// TwinCAT 3 PLC project Projet_Base
// ProgramVersion: 3.1.4022.3
// libraries:
//   Tc2_ControllerToolbox, * (Beckhoff Automation GmbH)
//   Tc2_IEC60870_5_10x, * (Beckhoff Automation GmbH)
//   Tc2_ModbusRTU, * (Beckhoff Automation GmbH)
//   Tc2_ModbusSrv, * (Beckhoff Automation GmbH)
//   Tc2_SerialCom, * (Beckhoff Automation GmbH)
//   Tc2_Standard, * (Beckhoff Automation GmbH)
//   Tc2_System, * (Beckhoff Automation GmbH)
//   Tc2_TcpIp, * (Beckhoff Automation GmbH)
//   Tc2_Utilities, * (Beckhoff Automation GmbH)
//   Tc3_Database, * (Beckhoff Automation GmbH)
//   Tc3_Module, * (Beckhoff Automation GmbH)
// project tree:
//   00_FunctionsBlocks/Beckhoff/AlarmManagement/ FB_HeartBeatMasterBackup.TcPOU (not stored), FUN_Alarms_CSV.TcPOU, FUN_ReadAlarm_CSV.TcPOU (not stored), ServerCSV.TcDUT, ServerSms.TcDUT, SMS_Server.TcPOU
//   00_FunctionsBlocks/Beckhoff/Annexesfunction/ FB_RestartService.TcPOU, FUN_ConnectVPN.TcPOU (not stored), FUN_DisconnectVPN.TcPOU (not stored), FUN_GetPublicIp.TcPOU (not stored), FUN_PingHost.TcPOU (not stored), PRG_RestartPlc.TcPOU (not stored)
//   00_FunctionsBlocks/Beckhoff/Communication/IEC104/ E_ComState.TcDUT (not stored), FB_IEC104ServerAkuo.TcPOU (not stored), GVL_Cst.TcGVL (not stored), ST_IEC104AkuoParam.TcDUT (not stored)
//   00_FunctionsBlocks/Beckhoff/Communication/Mail/ FUN_SendMail.TcPOU, ServerMail.TcDUT
//   00_FunctionsBlocks/Beckhoff/Communication/ModbusRTU/ CheckStruct.TcPOU (not stored), FB_ModbusRTU.TcPOU (not stored), FB_ReadModbusRTU_V2.TcPOU (not stored), Sample_ModbusRTU.TcPOU (not stored), Struct_InputRTU.TcDUT (not stored)
//   00_FunctionsBlocks/Beckhoff/Communication/ModbusTCP/ FB_ModbusRead.TcPOU (not stored), FB_ModbusReadCoils.TcPOU (not stored), FB_ModbusReadInput.TcPOU (not stored), FB_ModbusReadInputRegs.TcPOU (not stored), FB_ModbusWrite.TcPOU (not stored), FB_ModbusWriteMultipleCoils.TcPOU (not stored), FB_ModbusWriteSingleCoil.TcPOU (not stored), FB_ModbusWriteSingleRegister.TcPOU (not stored)
//   00_FunctionsBlocks/Beckhoff/Communication/SMS/ FB_DeleteAllSMS.TcPOU (not stored), FB_DeleteSMS.TcPOU (not stored), FB_Extract_Num_Mes.TcPOU (not stored), FB_Login.TcPOU (not stored), FB_ReadSMS.TcPOU (not stored), FB_SendSMS.TcPOU (not stored), ST_SMSDataSetEntry_Read.TcDUT (not stored), ST_SMSDataSetEntry_Send.TcDUT (not stored)
//   00_FunctionsBlocks/Beckhoff/Database/ CheckConfig.TcPOU (not stored), PRG_EpochConverter.TcPOU (not stored), PRG_TimestructConverter.TcPOU (not stored), St_DataHisto.TcDUT (not stored), St_DataHisto_Epoch.TcDUT (not stored), UnixTimestamp.TcPOU (not stored)
//   00_FunctionsBlocks/Beckhoff/Database/Firebird/ Firebird_CreateTables.TcPOU (not stored), Firebird_InsertBuffer.TcPOU (not stored), Firebird_InsertBuffer_vEpoch.TcPOU (not stored), Firebird_ReadAlarms.TcPOU (not stored), Firebird_RetrieveHDBID.TcPOU (not stored), Firebird_SelectBuffer.TcPOU (not stored), Firebird_WriteAlarms.TcPOU (not stored), LoggerFirebird.TcDUT (not stored), St_AlarmsV2.TcDUT (not stored)
//   00_FunctionsBlocks/Beckhoff/Database/InfluxDb/ InfluxDb_AlarmsManagement.TcPOU (not stored), InfluxDb_ReadValues.TcPOU (not stored), InfluxDb_WriteAlarms.TcPOU (not stored), InfluxDb_WriteStruct.TcPOU (not stored), LoggerInfluxDb.TcDUT (not stored), ST_InfluxAlarmsInsert.TcDUT (not stored), ST_InfluxAlarmsRetrieve.TcDUT (not stored)
//   00_FunctionsBlocks/Beckhoff/Database/SQLCe/ FB_SQLExpert_InsertBuffer_1.TcPOU (not stored)
//   00_FunctionsBlocks/Beckhoff/Database/SQLite/ SQLite_CreateDb_V2_1.TcPOU (not stored), SQLite_DeleteConfDb_1.TcPOU (not stored)
//   00_FunctionsBlocks/Beckhoff/DataProcessing/Compress/ FB_CompressFile.TcPOU (not stored), FUN_CompressCSV.TcPOU (not stored)
//   00_FunctionsBlocks/Beckhoff/DataProcessing/Database/ DataBase_V2.TcPOU (not stored), FB_DeleteFile.TcPOU (not stored), FB_SQLExpert_InsertBuffer.TcPOU (not stored), SQLite_CreateDb_V2.TcPOU (not stored), SQLite_DeleteConfDb.TcPOU (not stored)
//   00_FunctionsBlocks/Beckhoff/DataProcessing/ FB_MergeWordsToFloat.TcPOU (not stored), FB_MessageDynamique.TcPOU (not stored), FB_SplitFloatToWords.TcPOU (not stored), FB_WordsToFloat32MLE.TcPOU (not stored), FUN_Transpose.TcPOU (not stored), MOYENNE.TcPOU (not stored), ReplaceAll.TcPOU (not stored), SavePersistent.TcPOU (not stored)
//   00_FunctionsBlocks/Beckhoff/DataProcessing/ReadFile/ FB_Read.TcPOU (not stored), FB_ReadCSV.TcPOU (not stored)
//   00_FunctionsBlocks/Beckhoff/DataProcessing/WriteFile/ CheckStruct_Alarms.TcPOU (not stored), FB_CreateDir_V2.TcPOU (not stored), FB_WriteFile.TcPOU (not stored), FB_Write_CSV.TcPOU, FUN_CreateDir_CSV.TcPOU (not stored), LoggerCSV.TcDUT, ST_Journal.TcDUT (not stored), ST_ValuesAlarms.TcDUT (not stored), ST_ValuesWrite.TcDUT (not stored)
//   00_FunctionsBlocks/Beckhoff/Fifo/ FB_CommandAlternate.TcPOU (not stored), FB_DBDatasetFifo.TcPOU (not stored), FB_DBDatasetFifo_1min.TcPOU (not stored), FB_SMSDatasetFifo_Read.TcPOU (not stored), FB_SMSDatasetFifo_Send.TcPOU (not stored), GVL_Fifo.TcGVL (not stored)
//   00_FunctionsBlocks/Common/AlarmManagement/ FB_AlarmCodeManager.TcPOU (not stored), FB_CheckCommand.TcPOU (not stored), FB_CheckSetpt.TcPOU (not stored), FB_DetectFixedValue.TcPOU (not stored), FB_DetectFlicker.TcPOU (not stored), FB_UnknownEvent.TcPOU (not stored)
//   00_FunctionsBlocks/Common/BoolManagement/ FB_CountNinTimeWindow.TcPOU (not stored), FB_TapVariable.TcPOU (not stored), FB_Toggle2Tap.TcPOU (not stored), FB_WordToArrayOfBool.TcPOU (not stored), FB_WriteOnChange.TcPOU (not stored), RS_NoReset.TcPOU (not stored)
//   00_FunctionsBlocks/Common/Ctrl/ FB_PIDRegulation.TcPOU
//   00_FunctionsBlocks/Common/DataProcessing/ FB_Average.TcPOU (not stored), FB_CountBitOfWordAtTrue.TcPOU (not stored), FB_Integrate.TcPOU (not stored), FB_MovingAverage.TcPOU (not stored), FB_Ramp.TcPOU (not stored), FB_Ramp_Time.TcPOU (not stored), FB_Smooth.TcPOU (not stored), FB_XorWord.TcPOU (not stored), Split.TcPOU (not stored), Substring.TcPOU (not stored)
//   00_FunctionsBlocks/Common/DataProcessing/MergeWord/ FB_ISKRA_T5.TcPOU (not stored), FB_ISKRA_T6.TcPOU (not stored), FB_MergeWordsToDint.TcPOU (not stored), FB_MergeWordsToUint.TcPOU (not stored), FB_MergeWordsToUlint.TcPOU (not stored), FB_WordsToDint64BE.TcPOU (not stored)
//   00_FunctionsBlocks/Common/DataProcessing/SplitWord/ FB_SplitRealToWords.TcPOU (not stored), FB_SplitRealToWords_IEEE754.TcPOU (not stored), FB_SplitUlintToWords.TcPOU (not stored), FB_SplitWordToByte.TcPOU (not stored)
//   00_FunctionsBlocks/Common/HistorizationVisu/ FB_OperationIndex.TcPOU (not stored), GetTime.TcPOU (not stored)
//   00_FunctionsBlocks/Templates/ FB_EX_Example.TcPOU (not stored)
//   01_Equipement_Library/Actuators/ CB_Standard.TcDUT, CB_AuxMVCB_Sch.TcDUT, CB_FeederMVCB_Sch.TcDUT, CB_MainMVCB_Sch.TcDUT, CB_MeasureMVCB_Sch.TcDUT, FB_CB_GridMVCB.TcPOU, FB_CB_MainHVCB.TcPOU, FB_CB_MainMVCB.TcPOU, FB_CB_MeasureMVCB.TcPOU, CB_MainHVCB_Sch.TcDUT (not stored), CB.TcDUT, FB_CB_Base.TcPOU, FB_CB_AuxMVCB.TcPOU, FB_CB_FeederMVCB.TcPOU, FB_CB_MVSwitch.TcPOU
//   01_Equipement_Library/Datalogger/ Datalogger.TcDUT, Datalogger_IOWIT.TcDUT, Datalogger_SchSkid.TcDUT, Datalogger_Secu.TcDUT (not stored), Datalogger_SENECA.TcDUT (not stored), FB_Datalogger_Base.TcPOU, FB_Datalogger_IOWIT.TcPOU, FB_Datalogger_SchSkid.TcPOU, FB_Datalogger_SENECA.TcPOU, FB_Datalogger_PPCVerrerie.TcPOU, Datalogger_PPCVerrerie.TcDUT
//   01_Equipement_Library/GRID/ FB_GRID_Base.TcPOU, FB_GRID_Enedis.TcPOU, GRID.TcDUT, GRID_MADI.TcDUT (not stored), GRID_Enedis.TcDUT, FB_GRID_MADI.TcPOU, IEC104.TcDUT
//   01_Equipement_Library/Inverter/ FB_INV_Base.TcPOU, FB_INV_Smartlogger.TcPOU, FB_INV_Sun2000KtlMo.TcPOU, INV.TcDUT, INV_Huawei.TcDUT, SL_Huawei.TcDUT, STR.TcDUT
//   01_Equipement_Library/IPC/ FB_IPC.TcPOU, IPC.TcDUT
//   01_Equipement_Library/Operation Meter/ FB_PM_520x230.TcPOU, FB_PM_A40.TcPOU, FB_PM_Digiware.TcPOU, FB_PM_ION7650.TcPOU, FB_PM_Janitza.TcPOU, FB_PM_PM800.TcPOU, FB_PM_Q100.TcPOU, FB_PM_SM103E.TcPOU, PM.TcDUT, FB_PM_PM3250.TcPOU, PM_DirisA40.TcDUT (not stored), PM_Standard.TcDUT, PM_PM800.TcDUT (not stored), PM_Q100.TcDUT (not stored), FB_PM_Base.TcPOU
//   01_Equipement_Library/PCS/ DCInputs_PE.TcDUT (not stored), FB_PCS.TcPOU, FB_PCS_Base.TcPOU, FB_PCS_PE.TcPOU, PCS.TcDUT, PCS_Jema.TcDUT, PCS_PE.TcDUT, PowerCol_JemaAlarms.TcDUT, PowerCol.TcDUT, PowerCol_PE.TcDUT
//   01_Equipement_Library/ProtectRelay/ FB_ProtectRelay_DM2.TcPOU, FB_ProtectRelay_Flair23DM.TcPOU, FB_ProtectRelay_NSXCB.TcPOU, FB_ProtectRelay_PACE100ST.TcPOU, FB_ProtectRelay_REF615.TcPOU, FB_ProtectRelay_SepamT20.TcPOU, FB_ProtectRelay_VIP410.TcPOU, FB_ProtectRelay_WIP1.TcPOU, FB_ProtectRelay_SEPAM10a.TcPOU, FB_ProtectRelay_Base.TcPOU, FB_ProtectRelay_SepamS48.TcPOU, ProtectRelay_Standard.TcDUT (not stored), ProtectRelay_Flair23DM.TcDUT (not stored), ProtectRelay_NSXCB.TcDUT (not stored), ProtectRelay_PACE100ST.TcDUT (not stored), ProtectRelay_REFIO.TcDUT (not stored), ProtectRelay.TcDUT, ProtectRelay_S42.TcDUT (not stored), ProtectRelay_S48.TcDUT, ProtectRelay_T20.TcDUT (not stored), ProtectRelay_T87.TcDUT (not stored), ProtectRelay_VIP410.TcDUT (not stored), ProtectRelay_WIP1.TcDUT (not stored)
//   01_Equipement_Library/Router/ FB_Router.TcPOU, Router.TcDUT, Router_Standard.TcDUT
//   01_Equipement_Library/Sensors/ANA/ ANA_Standard.TcDUT, FB_ANA_IO.TcPOU, FB_ANA_Base.TcPOU, FB_ANA_Irra_Fx.TcPOU, ANA.TcDUT
//   01_Equipement_Library/Sensors/COM/ AllInOne.TcDUT, FB_AllInOne.TcPOU, FB_ANA_SMP1X.TcPOU, SMP1X.TcDUT
//   01_Equipement_Library/Sensors/TOR/ FB_TOR_CB.TcPOU, FB_TOR_Standard.TcPOU, FB_TOR_ES.TcPOU, FB_TOR_Fuse.TcPOU, FB_TOR_MS.TcPOU, FB_TOR_Spd.TcPOU, FB_TOR_VP.TcPOU, TOR.TcDUT, FB_TOR_Base.TcPOU, FB_TOR_DS.TcPOU, FB_TOR_Rain.TcPOU, FB_TOR_SD.TcPOU, FB_TOR_ToS.TcPOU, TOR_CB.TcDUT (not stored), TOR_Standard.TcDUT, TOR_Rain.TcDUT (not stored)
//   01_Equipement_Library/TAC/ FB_TAC.TcPOU (not stored), TAC.TcDUT (not stored), TAC_Standard.TcDUT (not stored)
//   01_Equipement_Library/Tariff Meter/ EM_Standard.TcDUT (not stored), FB_EM_Base.TcPOU, FB_EM_Pulse.TcPOU, EM.TcDUT (not stored)
//   01_Equipement_Library/Transfo/ FB_Transfo_Base.TcPOU, FB_Transfo_HVCom.TcPOU, FB_Transfo_MVCom.TcPOU, TapChanger.TcDUT (not stored), Transfo.TcDUT, FB_Transfo_MV.TcPOU, Transfo_HV.TcDUT (not stored), Transfo_MV.TcDUT
//   01_Equipement_Library/UPS/ FB_UPS_PS10048.TcPOU, UPS_CXC.TcDUT (not stored), FB_UPS_CXC.TcPOU, FB_UPS_Base.TcPOU, FB_UPS_Eneris.TcPOU, UPS.TcDUT, UPS_Eneris.TcDUT, UPS_PS10048.TcDUT (not stored)
//   02_Product_Library/PowerTRansformerStation%28PTR%29/ FB_PTR.TcPOU (not stored), FB_PTR_Base.TcPOU (not stored), PTR_Exd.TcDUT (not stored), PTR.TcDUT (not stored)
//   02_Product_Library/Substation%28SUB_MV%29/ FB_SUBMV.TcPOU (not stored), FB_SUBMV_Base.TcPOU (not stored), SUBMV.TcDUT (not stored), SUBMV_Exd.TcDUT (not stored)
//   02_Product_Library/WeatherStation %28WS%29/ FB_WS.TcPOU (not stored), FB_WS_Base.TcPOU (not stored), WS.TcDUT (not stored), WS_AGMA.TcDUT (not stored)
//   03_Power_Plant %28PP%29/ FB_PP.TcPOU (not stored), PP.TcDUT (not stored)
//   04_Application/ALARM/ FUN_Alarms.TcPOU, Redundancy.TcPOU (not stored)
//   04_Application/Annexes_Functions/ PRG_AnnexesFunctions.TcPOU
//   04_Application/BDD/ FUN_Write_CSV.TcPOU
//   04_Application/Checks/ CheckBounds.TcPOU (not stored), CheckDivDInt.TcPOU (not stored), CheckDivLInt.TcPOU (not stored), CheckDivLReal.TcPOU (not stored), CheckDivReal.TcPOU (not stored), CheckLRangeSigned.TcPOU (not stored), CheckLRangeUnsigned.TcPOU (not stored), CheckPointer.TcPOU (not stored), CheckRangeSigned.TcPOU (not stored), CheckRangeUnsigned.TcPOU (not stored)
//   04_Application/COM/ COM_Status.TcDUT (not stored), ModbusTcp.TcPOU (not stored)
//   04_Application/CONFIG/ GVL_BASE.TcGVL, GVL_Beckhoff.TcGVL (not stored), GVL_CFG.TcGVL, GVL_Check.TcGVL (not stored), GVL_DataBaseStructures.TcGVL (not stored)
//   04_Application/IO/ IO.TcDUT (not stored), PRG_IO.TcPOU, ST_AI.TcDUT, ST_AO.TcDUT, ST_DI.TcDUT, ST_DO.TcDUT
//   04_Application/MAIN/ MAIN.TcPOU, POU.TcPOU, TEST.TcPOU
//   04_Application/OPC/ AllDataR.TcDUT, AllDataWPulse.TcDUT, AllDataWToggle.TcDUT (not stored), AllValueW.TcDUT, OpcUa.TcPOU
//   / AnnexFunction.TcTTO, PlcTask.TcTTO
// real-time tasks:
//   TASK PlcTask: cycle T#10ms, priority 8, ADS port 350
//   TASK Emul_Task: cycle T#25000us, priority 16, ADS port 351
//   TASK Database_Task: cycle T#100000us, priority 14, ADS port 352
//   TASK IOTask: cycle T#10ms, priority 6, ADS port 301
//   TASK AnnexFunction: cycle T#100000us, priority 10, ADS port 353
// I/O:
//   DEVICE Périphérique 1 (EtherCAT) (disabled), AmsNetId 192.168.13.104.2.1
//     Terme 1 (EK1200) [EK1200-5000 EtherCAT Power supply (2A E-Bus)]
//       Terme 2 (EL4024) [EL4024 4Ch. Ana. Output 4-20mA, 12bit]
//       Terme 3 (EL3024) [EL3024 4Ch. Ana. Input 4-20mA DIFF]
//       Terme 4 (EL9011) [EL9011 End Terminal]

CONFIGURATION Projet_Base
    RESOURCE PLC ON TwinCAT3
        TASK AnnexFunction(INTERVAL := T#100000us, PRIORITY := 10);
        TASK PlcTask(INTERVAL := T#10ms, PRIORITY := 8);
        PROGRAM MAIN WITH PlcTask : MAIN;
        PROGRAM TEST WITH PlcTask : TEST;
    END_RESOURCE
END_CONFIGURATION

// ---- 00_FunctionsBlocks/Beckhoff/AlarmManagement/ServerCSV.TcDUT

TYPE ServerCSV :
STRUCT
	FileSize			: ULINT;			(*(o) Size of the file being used for logging alarms *)
	TimeCreation		: TIMESTRUCT;		(* TimeCreation of file*)
	TimeModif			: TIMESTRUCT;		(* Time Modif of file*)
	MesAlarmCode		: WORD;				(* Alarm Code related to this functionnality*)

END_STRUCT
END_TYPE

// ---- 00_FunctionsBlocks/Beckhoff/AlarmManagement/ServerSms.TcDUT

TYPE ServerSms :
STRUCT
	NbrUtiliActive			: INT;									(* Number of users*)
	MesAlarmCode			: WORD;									(* Alarm Code*)
	AX_Numtel				: ARRAY[1..CstNbUser] OF STRING(26);	(*Tel Number list*)
	AX_Subscribed			: ARRAY[1..CstNbUser] OF BOOL;			(*Subscription list*)
	AX_NomUtili				: ARRAY[1..CstNbUser] OF STRING(50); 	(* User name list	*)
	AX_UserLVL				: ARRAY[1..CstNbUser] OF WORD; 		(*User Level*)

END_STRUCT
END_TYPE

// ---- 00_FunctionsBlocks/Beckhoff/Communication/Mail/ServerMail.TcDUT

TYPE ServerMail :
STRUCT

	MesAlarmCode			: WORD;			(*alarm code *)
	
	AX_MailAddr				: ARRAY[1..CstNbUser] OF STRING(255);		(* Mail Address List*)
	AX_Subscribed			: ARRAY[1..CstNbUser] OF BOOL;				(* Mail subscription list*)
	AX_NomUtili				: ARRAY[1..CstNbUser] OF STRING(50); 		(* User Name List*)
	AX_UserLVL				: ARRAY[1..CstNbUser] OF WORD; 		(* User Level*)
	
	OUT_NbMailSent			: ULINT;									(* Number of mail being sent *)
	
END_STRUCT
END_TYPE

// ---- 00_FunctionsBlocks/Beckhoff/DataProcessing/WriteFile/LoggerCSV.TcDUT

TYPE LoggerCSV :
STRUCT
	FileSize			: ULINT;			(* (o) File size *)
	TimeCreation		: TIMESTRUCT;		(* TimeCreation of file*)
	TimeModif			: TIMESTRUCT;		(* Time Modif of file*)
	MesAlarmCode		: WORD;				(* Alarm Code*)

END_STRUCT
END_TYPE

// ---- 01_Equipement_Library/Actuators/CB_Standard.TcDUT
TYPE CB_Standard :
///////////
// Structure For Bousquet. Main Operating Data to be saved ( ex: OPC )   
//////////
STRUCT
	//DI
	MesData				: CB ;  (* Object*)

END_STRUCT
END_TYPE

// ---- 01_Equipement_Library/Actuators/CB_AuxMVCB_Sch.TcDUT
///////////
// Structure For Bousquet. Main Operating Data to be saved (ex: OPC).  
//////////

TYPE CB_AuxMVCB_Sch :
STRUCT
	//DI
	MesData					: CB ;      (* Object*)
	MesFuseBurned		    : BOOL ; 	(* The Fuse is burned*)
	MesEarth				: BOOL ; 	(* The Cell is grounded*)

END_STRUCT
END_TYPE

// ---- 01_Equipement_Library/Actuators/CB_FeederMVCB_Sch.TcDUT
///////////
// Structure For Bousquet . Main Operating Data to be saved (ex: OPC).  
//////////

TYPE CB_FeederMVCB_Sch :
STRUCT
	//DI
	MesData					: CB   ;    (* Object*)
	MesComutLocal		    : BOOL ; 	(* The cell selector is in local position*)
	MesAlarmPwr		        : BOOL ; 	(* The cell motorization has a power supply fault*)
	MesEarth				: BOOL ; 	(* The cell is grounded (earthing)*)
	MesTripped	    	    : BOOL ; 	(* The cell is tripped (opened and locked due to alarm)*)
	OUT_CmdOpen				: BOOL ; 	(* The SCADA sends an Open command to the cell*)
	OUT_CmdClose			: BOOL ; 	(* The SCADA sends a Close command to the cell*)
	MesOpened_Sect			: BOOL ;    (* The associated switchgear is opened*)
	
END_STRUCT
END_TYPE

// ---- 01_Equipement_Library/Actuators/CB_MainMVCB_Sch.TcDUT
///////////
// Structure for MainMVCB Schneider. Main Operating Data to be saved (ex: OPC).  
//////////

TYPE CB_MainMVCB_Sch :
STRUCT
	//DI
	MesData					: CB   ;    (* Object*)
	MesComutLocal		    : BOOL ; 	(* The cell selector is in local position*)
	MesAlarmPwr		        : BOOL ; 	(* The cell motorization has a power supply fault*)
	MesEarth				: BOOL ; 	(* The cell is grounded (earthing)*)
	MesTripped	    	    : BOOL ; 	(* The cell is tripped (opened and locked due to alarm)*)
	OUT_CmdOpen				: BOOL ; 	(* The SCADA sends an Open command to the cell*)
	OUT_CmdClose			: BOOL ; 	(* The SCADA sends a Close command to the cell*)
	MesOpened_Sect			: BOOL ; 	(* The associated switchgear is opened*)
	
END_STRUCT
END_TYPE

// ---- 01_Equipement_Library/Actuators/CB_MeasureMVCB_Sch.TcDUT
///////////
// Structure For Bousquet. Main Operating Data to be saved (ex: OPC).  
//////////

TYPE CB_MeasureMVCB_Sch :
STRUCT
	//DI
	MesData					: CB ;      (* Object*)
	MesFuseBurned		    : BOOL ; 	(* The Fuse is burned*)
	MesEarth				: BOOL ; 	(* The Cell is grounded*)

END_STRUCT
END_TYPE

// ---- 01_Equipement_Library/Actuators/CB.TcDUT
TYPE CB :
///////////
// Structure For Bousquet. Main Operating Data to be saved ( ex: OPC )   
//////////
STRUCT
	//DI
	MesClosed		: BOOL ;	(* Cell is closed*)
	MesOpened		: BOOL ;	(* cell is opened*)
	
	MesAlarmCode	: WORD ;	(* Internal Akuo Alarm Code*)
	MesWarningCode	: WORD ;	(* Internal Akuo Warning Code*)
	MesEventCode	: WORD ;	(* Internal Akuo Warning Code*)
	
	MesCP_Open		: BOOL ;   	(* Cal(NA) Permanent Conditions*)
	MesCP_Close		: BOOL ; 	(* Cal(NA) Permanent Conditions*) 

END_STRUCT
END_TYPE

// ---- 01_Equipement_Library/Datalogger/Datalogger.TcDUT
TYPE Datalogger :
STRUCT
	MesAlarmCom					: BOOL ; 						(* (NA) Communication alarm *)
	MesAlarmCode				: WORD ; 						(* (NA) Internal Akuo Alarm Code				*)
	MesWarningCode				: WORD ; 						(* (NA) Internal Akuo Warning Code       	*)
	MesEventCode				: WORD ; 						(* (NA) Internal Akuo Event Code         	*)
	 
	MesCP_Read					: BOOL; 						(* (NA) Permanent conditions for read		*)          

	MesCP_Write					: BOOL; 						(* (NA) Permanent conditions for read		*)    
                             						
END_STRUCT
END_TYPE

// ---- 01_Equipement_Library/Datalogger/Datalogger_IOWIT.TcDUT
TYPE Datalogger_IOWIT :		// Data from WIT in PTR
STRUCT
	

	MesData						: Datalogger ; 
		            			
	Transfo						: Transfo_MV ; 
	                			
	WS							: WS_PTR ; 
	                			
	MainMVCB					: MainMVCB_Sch ; 
	CB_INV						: ARRAY[1..CstNbInv_PTR_G] OF  TOR ; 
	CB_Transfo					: TOR ; 
	                				
	FSS							: FSS ; 
	DS							: TOR ; 
	MS	 						: TOR ; 





	MesInvReturnContact1 		: BOOL;		(* Inverter return contact 1 *)
	MesInvReturnContact2 		: BOOL;		(*  Inverter return contact 2 *)
	MesTransfoLocalTemp			: REAL;		(* (°C) Transformer room temperature *)
	
	MesCP_Read					: BOOL; 	(* permanent conditions for read *)

	MesAlarmCode				: WORD ; 	(* Internal Akuo Alarm Code *)
	MesWarningCode				: WORD ; 	(* Internal Akuo Warning Code *)
	MesEventCode				: WORD ; 	(* Internal Akuo Event Code *)
END_STRUCT
END_TYPE

// ---- 01_Equipement_Library/Datalogger/Datalogger_SchSkid.TcDUT
TYPE Datalogger_SchSkid :
STRUCT

	MesData							: Datalogger ; 							(* MesData *)
                        			                			
	MesComutLocal					: BOOL; 								(* FALSE := Local, TRUE := Remote (DI_204) *)
	MesState_MVCB					: BOOL; 								(* True := Fermé, False := Ouvert (DI_205) *)
	MesWatchdog_ProtectRelayVIP		: BOOL; 								(* WatchDog of VIP410 (DI_201)			   *)
	MesFault_ProtectRelayVIP		: BOOL; 								(* TRUE:= Fault, False:= OK, Déclenchement du défaut VIP (DI_206) *)
	                        			
	MesToggleRead					: BOOL; 								(* Cal State com of FB IO *)
	MesToggleWrite					: BOOL;;  								(* Cal State com of FB IO *)
	 
	DS_Synthesis					: TOR ; 								(* Synthesis of door sensors True = a door is opened (DI_209) 			 *)
	CB_INV							: ARRAY[1..CstNbInv_PTR_G] OF  TOR; 	(* TRUE := CB opened, False : CB closed, INV 1 (DI_202) / INV 2 (DI_203) *)
	Transfo_Synthesis				: Transfo_MV; 							(* Transfo *)
	 	 						
END_STRUCT
END_TYPE

// ---- 01_Equipement_Library/GRID/GRID.TcDUT
///////////
// Structure For DEIECommand. Main Operating Data to be saved (ex: OPC)  
//////////
TYPE GRID :
STRUCT
	// TC
	OUT_CmdAutCpl			 	: BOOL ;			(* (NA) Autorisation couplage (pulse)*)
	OUT_CmdDisconnect		 	: BOOL ;			(* (NA) Disconnect command (pulse)*)
	OUT_CmdEmergencyDisconnect	: BOOL ;			(* (NA) Emergency disconnect command (pulse)*)	
	OUT_SetptP 				 	: REAL ;			(* (kW) P Setpoint from EDF*)
	OUT_SetptQ 				 	: REAL ;			(* (kVar) Q Setpoint from EDF*)
	OUT_MesPPUnavailable		: BOOL ;			(* (NA) TS centrale indisponible*)
	OUT_MesPPConnected			: BOOL ; 			(* (NA)Centrale couplée(1)/Centrale Découplée(0)*)	
	
	// State 	
	MesAlarmCode				: WORD ; 			(* (NA) Internal Akuo Alarm Code*)
	MesWarningCode 			 	: WORD ; 			(* (NA) Internal Akuo Warning Code*)
	MesEventCode			 	: WORD ;			(* (NA) Internal Akuo Warning Code*)
	MesEventCode2				: WORD ; 			(* (NA) EventCode 2*)

	MesAlarmCom				 	: BOOL ;			(* (NA) Communication alarm *)
	MesCP_Read				 	: BOOL := TRUE; 	(* (NA) Cal : Read function enable*)
	
END_STRUCT
END_TYPE

// ---- 01_Equipement_Library/GRID/GRID_Enedis.TcDUT
///////////
// Structure For DEIECommand. Main Operating Data to be saved (ex: OPC).
//////////
TYPE GRID_Enedis :
STRUCT
	
	MesData								: GRID ; 		(* GRID MesData *)
                                       	
	OUT_CmdPReg                         : BOOL ;     	(* (NA) Passage à P0 reçu DI*)
	OUT_CmdQReg	                   	    : BOOL ;     	(* (NA) Passage à Q0 reçu DI*)

	OUT_Rse								: BOOL; 		(* (NA) Protection en Rse(1) / Protection Hors RSE (O) *)
	OUT_TA								: BOOL; 		(* (NA) Telecaction en service (1) / Teleaction Hors service (0)*)
	
END_STRUCT
END_TYPE

// ---- 01_Equipement_Library/GRID/IEC104.TcDUT
///////////
// Structure For DEIECommand. Main Operating Data to be saved ( ex: OPC ) .  
//////////
TYPE IEC104 :
STRUCT

	(* Memory offset 0..99 unused *)
	(* Single points *)// MAx 8 bit per register . 0..7
	OUT_MesLocal			AT%MX10.0 	: BOOL;			(* IOA 12 BAT.LOCAL*)
	OUT_MesModeManuel_on	AT%MX10.1 	: BOOL; 		(* IOA 13 MANUAL*)
	OUT_MesModeAuto_on		AT%MX10.2 	: BOOL; 		(* IOA 14 AUTO*)
	OUT_MesCharging			AT%MX10.3 	: BOOL;			(* IOA 15 CHARGE.BAT*)
	OUT_MesDischarging		AT%MX10.4 	: BOOL;			(* IOA 16 DESCHARGE.BAT*)
	OUT_MesEs				AT%MX10.5 	: BOOL; 		(* IOA 20 ARRET.URGENCE*)
	OUT_MesToS				AT%MX10.6 	: BOOL; 		(* IOA 21 PRESENCE*)
	OUT_MesIncident			AT%MX10.7 	: BOOL;			(* IOA 19 INCIDENT*)
	OUT_MesFaultTeleMes		AT%MX11.0 	: BOOL;			(* IOA 37 DEFAUT CARTE TM*)
	OUT_MesFaultTeleCmd		AT%MX11.1 	: BOOL;			(* IOA 38 DEF FUNC TC*)
	OUT_MesFaultTeleSgnl	AT%MX11.2 	: BOOL;			(* IOA 39 DEF FONC TS*)
	OUT_MesIECServerFault	AT%MX11.3 	: BOOL;			(* IOA 41 DEF LIAISON 104*)
	
	(* Double points *)
	(* 	Bit 0..1 = MesStartOn,
		Bit 2..3 = MesComTest_ON, 
		Bit 4..5 = MesCentraleCpl, 
		Bit 6..7 = MesCentrale_Ind*)
	OUT_MesDouble			AT%MB12		: BYTE;
	MesDJOpen							: BOOL; 		(* IOA 51 DJ OPEN*)
	MesSoutirage_on						: BOOL;			(* IOA 43 ARRET.BAT*)
	MesComTest_on						: BOOL; 		(* IOA 44 TC.SOUTIRAGE *)
	MesCentrale_Cpl						: BOOL;			(* IOA 17 COUPL*)
	MesCentrale_indispo					: BOOL;			(* IOA 22 DISPO*)
	
	(* Measured values, short floating point values *)
	OUT_MesEconnected 		AT%MB42		: REAL;			(*IOA 5 NIVEAU BAT*)
	OUT_MesEmaxconnected 	AT%MB14		: REAL; 		(*IOA 6 STOCK MAX*)
	OUT_MesP 				AT%MB18		: REAL; 		(*IOA 1 P.ACTIVE*)
	OUT_MesQ 				AT%MB22		: REAL; 		(*IOA 2 P.REACTIVE*)
	OUT_MesU_HTA 			AT%MB26		: REAL; 		(*IOA 3 U.HTA*)
	OUT_MesFreq 			AT%MB30		: REAL; 		(*IOA 4 FREQUENCE*)
	OUT_MesPdispo_inj 		AT%MB34		: REAL; 		(*IOA 7 P.INJ MAX*)
	OUT_MesPdispo_abs 		AT%MB38		: REAL; 		(*IOA 8 P.SOUT MAX*)

	(*#################################################################*)
	(* TC *)
	IN_CmdModeManuel		AT%MX60.0 	: BOOL;			(* IOA 30 TC.MANUEL*)
	IN_CmdModeManuelOff		AT%MX60.1 	: BOOL;			(* Not implemented yet*)
	IN_CmdAut_Cpl			AT%MX60.2 	: BOOL; 		(* IOA 32 TC.COUPLAGE*)
	IN_CmdDisconnect		AT%MX60.3 	: BOOL;			(* IOA 33 TC.DECOUPLAGE*)
	IN_CmdConnect			AT%MX60.4 	: BOOL;			(* Not implemented*)
	
	(* TCD *)
	(* 	Bit 0..1 = command disconnecr,
		Bit 2..3 = command start, 
		Bit 4..5 =  command test, 
		Bit 6..7 = fourth double command *)
	IN_Cmddouble			AT%MB61		: BYTE;			(**)
	CmdSoutirage						: BOOL;			(* IOA 26 soutirage*)
	CmdTest								: BOOL;			(* IOA 27 TC.FICTIVE*)

	//TVC
	IN_SetptP 				AT%MB72 	: REAL ;		(*IOA 36 CONSIGNE P*)
	IN_ParamPmax 			AT%MB64 	: REAL ;    	(*IOA 34 CONSIGNE P+MAX *)
	IN_ParamPmin 			AT%MB68 	: REAL ;		(*IOA 35 CONSIGNE P-MAX *)

	
END_STRUCT
END_TYPE

// ---- 01_Equipement_Library/Inverter/INV.TcDUT
///////////
// Structure For Inverter. Main Operating Data to be saved (ex: OPC).  
//////////
TYPE INV :
STRUCT
	
		// INV Measures from Datalogger
		MesP 				: REAL ; 		(* (kW) 	Active Power output (AC) of inverter PCS01*)
		MesQ 				: REAL ;  		(* (kVAr)   Reactive AC Power Produced				  *)
		MesPdc 				: REAL ;  		(* (kW) 	Power measure (DC) of inverter			  *)
		MesIdc 				: REAL ;	 	(* (A) 	    Total Current measure (DC)				  *)
		MesUdc 				: REAL ;  		(* (V)  	Mean Voltage measure (DC)				  *)
		MesU 				: REAL ;		(* (V) 	    Mean Voltage measure (AC)				  *)
		MesV				: REAL ; 		(* (V)      Mean Phase to Neutral voltage			  *)
		MesI				: REAL ;		(* (A)      Mean Phase Current						  *)
		MesI0               : REAL ;        (* (A) 		Residual current						  *) 
		MesFreq				: REAL ; 		(* (Hz)     Frequency                                 *)
		MesS				: REAL ; 		(* (kVA)     Apparent Power						      *)
		MesInsuResistor		: REAL ; 		(* (MOhms) Insulation Resistance					  *)
		MesCosPhi			: REAL ; 		(* (p.u) Power Factor								  *)
		MesTemp				: REAL ; 		(* (C) Inverter Temperature							  *)
		MesState_Inv			: UINT ;		(* (NA) Inverter Status								  *)
		ParamPn				: REAL ; 		(* (kW) Nominal Capacity of SMA 25000 TL Inverter	  *)
		ParamQn				: REAL ;		(* (kVAr) Nominal reactive power 					  *)
		MesCurtl		    : BOOL ; 		(* (NA)Cal True if the inverter is curtailing Power	  *)
		MesAlarmCom			: BOOL ; 		(* (NA) Communication Alarm							  *)
		MesCP_Read			: BOOL := TRUE;	(* (NA) Cal : Permanent Condition for Read			  *)
		MesCP_Write			: BOOL := FALSE;	(* (NA) Cal : Permanenent Condition for Write		  *)
		                                                                                        
		MesOpened_Ac        : BOOL ;   		(* (NA) Ac switch is opened							  *)
		MesOpened_Dc        : BOOL ;   		(* (NA) Dc switch is opened							  *)
		                                                                                        
		OUT_CmdStart        : BOOL ;        (* (NA) OUT start command 							  *)
		OUT_CmdStop         : BOOL ;        (* (NA) OUT stop command   							  *)
		OUT_SetptPLimit    	: REAL ;        (* (kW) OUT P setpoint  							  *)
		OUT_SetptQ          : REAL ;        (* (kVAr)  OUT Q setpoint   						  *)
		MesIDState			: WORD ; 		(* (NA) Cal: Akuo Internal State . O=Stopped, 1 = RUN, 2 = Curtailment *)
		MesAlarmCode		: WORD ; 		(* (NA) Internal Akuo AlarmCode                       *)
		MesWarningCode		: WORD ; 		(* (NA) Internal Akuo WarningCode                     *)
		MesEventCode		: WORD ; 		(* (NA) Internal Akuo EventCode                       *)

END_STRUCT
END_TYPE

// ---- 01_Equipement_Library/Inverter/INV_Huawei.TcDUT
///////////
// Structure For Inverter. Main Operating Data to be saved ( ex: OPC ) .  
//////////
TYPE INV_Huawei :
STRUCT
	
	// INV Measures
		MesData			: INV ; (* INV *) 

		STR				: ARRAY[1..12 ] OF STR ;  	(* STR *) 
		
		MesEDay			: REAL ;	    			(* (kWh)Daily Energy	*)
	    MesETot			: REAL ;					(* (kWh)Total Energy	*)
		MesI1			: REAL ;					(*	(A) MesI1			*)
		MesI2			: REAL ;					(*	(A) MesI2			*)
	    MesI3			: REAL ;					(*	(A) MesI3			*)
		MesU12			: REAL ;					(*	(V) MesU12			*)
        MesU23			: REAL ;					(*	(V) MesU23			*)
        MesU31			: REAL ;					(*	(V) MesU31			*)
		MesV1			: REAL ;					(*	(V) MesV1			*)
		MesV2			: REAL ;					(*	(V) MesV2			*)
		MesV3			: REAL ;					(*	(V) MesV3			*)
                                        			
		MesStateIndic 	: WORD ;					(*	MesStateIndic 		*)
		MesOpeStatus 	: WORD ;					(*	MesOpeStatus 		*)
		MesAlm1			: WORD ;					(*	MesAlm1				*)
		MesAlm2			: WORD ;					(*	MesAlm2				*)
		MesAlm3			: WORD ;					(*	MesAlm3				*)

END_STRUCT
END_TYPE

// ---- 01_Equipement_Library/Inverter/SL_Huawei.TcDUT
///////////
// Structure For Inverter. Main Operating Data to be saved ( ex: OPC ) .  
//////////
TYPE SL_Huawei :
STRUCT
	
		MesData				: INV ;  (* INV *) 
	
	// INV Measures
		MesEDay				: REAL ;     	(*/ (kWh) Daily Energy*)
	    MesETot				: REAL ;		(*/ (kWh) Total Energy*)
		MesOn				: BOOL ;        (* Smartlogger is ON*)
		MesI1				: REAL ;        (* (A) AC current phase 1*)
		MesI2				: REAL ;        (* (A) AC current phase 1*)
	    MesI3				: REAL ;        (* (A) AC current phase 1*)
		MesU12				: REAL ;        (*(V) AC Voltage phase1 to phase2*)
        MesU23				: REAL ;        (*(V) AC Voltage phase2 to phase3*)
        MesU31				: REAL ;        (*(V) AC Voltage phase3 to phase1*)
		MesEff				: REAL ; 		(* (%) Inverter efficiency*)
		MesSetptPMax		: REAL ;        (* (kW) Maximal Active power setpoint*)
		MesSetptQMax		: REAL ;        (*(kVAr) Maximal reactive power setpoint*)
		MesSetptQMin		: REAL ;        (*(kVAr) Minimal reactive power setpoint*)
		OUT_SetptPlimit		: REAL ;        (*(kW) Maximal Active power setpoint sent by PPC*)
		OUT_SetptQlimit		: REAL ;        (*(kVAr) Maximal Reactive power setpoint sent by PPC*)

END_STRUCT
END_TYPE

// ---- 01_Equipement_Library/Inverter/STR.TcDUT
TYPE STR :
STRUCT
		MesIdc			: REAL;   						(* (A) DC current *)
		MesUdc			: REAL;							(* (V) DC voltage *)
END_STRUCT
END_TYPE

// ---- 01_Equipement_Library/IPC/IPC.TcDUT
TYPE IPC :
STRUCT
		
		MesAlarmCode		: WORD ;	(* (NA) Internal Akuo AlarmCode		*)
		MesWarningCode		: WORD ; 	(* (NA) Internal Akuo WarningCode   *)
		MesEventCode		: WORD ; 	(* (NA) Internal Akuo EventCode	    *)
		
END_STRUCT
END_TYPE

// ---- 01_Equipement_Library/Operation Meter/PM.TcDUT
///////////
// Structure For I35. Main Operating Data to be saved (ex: OPC).  
//////////
TYPE PM :
STRUCT
		MesU12						: REAL ; (* (V) Phase1 - Phase 2 AC Voltage 		   			*)
		MesU23						: REAL ; (* (V) Phase2 - Phase 3 AC Voltage         			*)
		MesU31						: REAL ; (* (V) Phase3 - Phase 1 AC Voltage         			*)
  		MesV1						: REAL ; (* (V) Phase1 AC Voltage                   			*)
		MesV2						: REAL ; (* (V) Phase2 AC Voltage                   			*)
		MesV3						: REAL ; (* (V) Phase3 AC Voltage		           				*)
		MesFreq						: REAL ; (* (Hz)Frequency		                   				*)
		MesI1						: REAL ; (* (A) AC current Phase 1                  			*)
		MesI2						: REAL ; (* (A) AC current Phase 2                  			*)
		MesI3						: REAL ; (* (A) AC current Phase 3                  			*)
		MesIn						: REAL ; (* (A) Neutral AC current                  			*)
		MesP						: REAL ; (* (kW) Total Active power                 			*)
		MesQ						: REAL ; (* (kVAr) Total Reactive Power Phase 1     			*)
		MesS						: REAL ; (* (kVA)Total Apparent power		       				*)
		MesCosPhi					: REAL ; (* (NA) Power factor                       			*)
		MesP1						: REAL ; (* (kW) Active Power Phase 1               			*)
		MesP2						: REAL ; (* (kW) Active Power Phase 2               			*)
		MesP3						: REAL ; (* (kW) Active Power phase 3               			*)
		MesQ1						: REAL ; (* (kVAr)Reactive Power Phase 1            			*)
		MesQ2						: REAL ; (* (kVAr)Reactive Power Phase 2            			*)
		MesQ3						: REAL ; (* (kVAr)Reactive Power Phase 3            			*)
		MesS1						: REAL ; (* (kVA) Total Apparent power Phase 1      			*)
		MesS2						: REAL ; (* (kVA) Total Apparent power Phase 2      			*)
		MesS3						: REAL ; (* (kVA) Total Apparent power Phase 3      			*)
		MesEActCons					: REAL ; (* (kWh) Recieved active energy            			*)
		MesEReactCons				: REAL ; (* (kVArh) 	Recieved reactive energy       			*)
		MesEActProd					: REAL ; (* (kWh) Delivered active energy           			*)
		MesEReactProd				: REAL ; (* (kVArh) 	Delivered reactive energy	   			*)
		MesI						: REAL ; (* (A) Mean AC current                     			*)
		MesV						: REAL ; (* (V) Mean Simple Phase AC Voltage        			*)
		MesU						: REAL ; (* (V) Mean Phase - Phase  AC Voltage      			*)
		MesCosPhi1                  : REAL ; (* (NA) Total Power Factor Phase 1         			*)
		MesCosPhi2                  : REAL ; (* (NA) Total Power Factor Phase 2         			*)
		MesCosPhi3                  : REAL ; (* (NA) Total Power Factor Phase 3         			*)
		MesTanPhi					: REAL ; (* (NA) Total Tangeante phi                			*)

		MesAlarmCom					: BOOL ;  		 (* (NA) Communication Error with I35 module    *)
		MesCP_Read					: BOOL := TRUE ; (* (NA) Cal: Read FUNCTION enable 				*)
		                                                                                        	
		MesAlarmCode				: WORD ; (* (NA) Internal Akuo Alarm Code			   			*)
		MesWarningCode				: WORD ; (* (NA) Internal Akuo Warning Code			  			*)
END_STRUCT
END_TYPE

// ---- 01_Equipement_Library/Operation Meter/PM_Standard.TcDUT
///////////
// Structure For I35. Main Operating Data to be saved (ex: OPC).  
//////////
TYPE PM_Standard :
STRUCT
		MesData						: PM ; (* Object *) 
	
END_STRUCT
END_TYPE

// ---- 01_Equipement_Library/Datalogger/Datalogger_PPCVerrerie.TcDUT
TYPE Datalogger_PPCVerrerie :
STRUCT
	MesData			: Datalogger ; 

	
	//225 kV 
//	PM_225kV									: PM ; // ION non remonté 
                                    			
	ProtectRelay_MainHVCB						: ProtectRelay_S42 ; 
	MainHVCB									: CB_MainHVCB_Sch ; 
                                    			
//	A1_GridHVCB									: GridHVCB ; Non remonté ? 
                                    			
	ProtectRelay_Transfo225kV					: ProtectRelay_T87 ; 
	Transfo_225kV								: Transfo_HV ; 	
	GRID										: GRID ; // non remonté ? 
	                                			
	                                			
                                    			
//	20 kV 		                    			
	MainMVCB									: MainMVCB_Sch ; 
	ProtectRelay_MainMVCB						: ProtectRelay_S42 ; 
						            			
	ProtectRelay_FeederMVCB						: ARRAY[1..2] OF ProtectRelay_S42 ; 		// 1. Midi 2. Plat 
	FeederMVCB									: ARRAY[1..2] OF FeederMVCB_Sch ; 
	                                	
                                    	
	                                	
	// Aux                          	
	Transfo_Aux									:  Transfo_MV ; 
	                                			
	UPS_CE										: UPS_VERR ; 
	UPS_TCM										: UPS_VERR ; 
	TapChanger 									: TapChanger ; 
	FSS											: FSS; 				(*Fire System*)
	DS											: TOR ; 			(*Door Sensor*)
	ES											: TOR ; 			(*Emergency Stop*)
	

	// Substation
	MesState									: WORD ; 			// Calculated  State of the HV + MV substation. 


	                                    		                   
	// 20 kV Courant Neutre et Cuve                                
    // transfo          ?????                                                    
	Mes20kVCourNeutCuveDefaultMasseCuve1		: BOOL;            	(*CourNeutCuveDefaultMasseCuve1	 	 *)
	Mes20kVCourNeutCuveMaxIexp2					: BOOL;            	(*CourNeutCuveMaxIexp2				 *)
	Mes20kVCourNeutCuveDefaultMasseCuve2		: BOOL;            	(*CourNeutCuveDefaultMasseCuve2	 	 *)
	Mes20kVCourNeutCuveMaxIexp4					: BOOL;            	(*CourNeutCuveMaxIexp4				 *)
	Mes20kVCourNeutCuveDefaultGround			: BOOL;            	(*CourNeutCuveDefaultGround		 	 *)
	Mes20kVCourNeutCuveMaxI0exp4				: BOOL;            	(*CourNeutCuveMaxI0exp4			 	 *)
	Mes20kVCourNeutCuveTempAlarm				: BOOL;            	(*CourNeutCuveTempAlarm			 	 *)
	Mes20kVCourNeutCuveTempTrigger				: BOOL;            	(*CourNeutCuveTempTrigger			 *)
	Mes20kVCourNeutCuveGazDischarge				: BOOL;            	(*CourNeutCuveGazDischarge			 *)
	Mes20kVCourNeutCuvePressure					: BOOL;   		   	(*CourNeutCuvePressure				 *)
	                                    		                   	
	Mes20kVCourNeutCuveI1						: REAL;            	(*(A) CourNeutCuveI1			 *)
	Mes20kVCourNeutCuveResidualI				: REAL;            	(*(A) CourNeutCuveResidualI	     *)
	Mes20kVCourNeutCuveDecltI1					: REAL;            	(*(A) CourNeutCuveDecltI1		 *)
	Mes20kVCourNeutCuveDecltI2					: REAL;            	(*(A) CourNeutCuveDecltI2		 *)
	                                                               	
	// Aux HT, BT and Transfo                                      	
	 // AuxMVCB                                                    	          
	MesAuxHTSect225kV							: BOOL;		       	(* AuxHTSect225kV						*)
	MesAuxHtSmaltHTBOpen						: BOOL;		       	(* AuxHtSmaltHTBOpen					*)
	MesAuxHtFusionFuseMeasures225kV				: BOOL;		       	(* AuxHtFusionFuseMeasures225kV			*)                                              
	MesAuxHtFusionFuseProtect225kV				: BOOL;		       	(* AuxHtFusionFuseProtect225kV			*)
	MesAuxHtFusionFuseCountRte225kV				: BOOL;		       	(* AuxHtFusionFuseCountRte225kV			*)
	MesAuxHtShortCircuitCurrentProtectCcp2		: BOOL;		       	(* AuxHtShortCircuitCurrentProtectCcp2	*)
	MesAuxHtDisjCount20kVOpen					: BOOL;		       	(* AuxHtDisjCount20kVOpen				*)
	MesAuxHtDisjRefVoltage20kVOpen				: BOOL;		       	(* AuxHtDisjRefVoltage20kVOpen			*)
	MesAuxHtShortCircuitCurrentProtectCcp3		: BOOL;		       	(* AuxHtShortCircuitCurrentProtectCcp3	*)
                                                                   	
	MesAuxBtTriggerGeneralDisj					: BOOL;		       	(*AuxBtTriggerGeneralDisj				 *)
	MesAuxBt400VManqueAC						: BOOL;		       	(*AuxBt400VManqueAC					     *)
	MesAuxBt400VDecltAntenneScada				: BOOL;		       	(*AuxBt400VDecltAntenneScada			 *)
	MesAuxBt400VDecltAntennePrio				: BOOL;		       	(*AuxBt400VDecltAntennePrio			 	 *)
	MesAuxBt400VPermutAutoStopMode				: BOOL;		       	(*AuxBt400VPermutAutoStopMode			 *)
	MesAuxBt400VPermutAutoNormalMode			: BOOL;		       	(*AuxBt400VPermutAutoNormalMode		 	 *)
	MesAuxBt400VPermutAutoSecoursMode			: BOOL;		       	(*AuxBt400VPermutAutoSecoursMode		 *)
	MesAuxBt400VPermutModeAuto					: BOOL;    	       	(*AuxBt400VPermutModeAuto				 *)
	MesAuxBt400VVoltageLossNormalAlim			: BOOL;		       	(*AuxBt400VVoltageLossNormalAlim		 *)
	MesAuxBt400VVoltageLossSecoursAlim			: BOOL;		       	(*AuxBt400VVoltageLossSecoursAlim		 *)
	MesAuxBt400VDefaultPermut					: BOOL;		       	(*AuxBt400VDefaultPermut				 *)


	MesAuxBtDefaultInverter						: BOOL;  		   	(* AuxBtDefaultInverter	*)
                                                                   	
	MesAuxBtSyntDefaultDistrib48VccJdb			: BOOL;  		   	(* AuxBtSyntDefaultDistrib48VccJdb		*)
	MesAuxBtSyntOpenDistrib48VccJdb				: BOOL;		       	(* AuxBtSyntOpenDistrib48VccJdb			*)
	MesAuxBtSyntDefaultDistrib48VccLocker		: BOOL;  		   	(* AuxBtSyntDefaultDistrib48VccLocker	*)
    MesAuxBtSyntOpenDistrib48VccLocker			: BOOL;		       	(* AuxBtSyntOpenDistrib48VccLocker		*)
                                                                   	
	MesAuxTransfoMeltingFusesContact			: BOOL;		       	(* AuxTransfoMeltingFusesContact	*)
                                                                   	
	MesAuxTransfoSwitchGear						: BOOL;	           	(*AuxTransfoSwitchGear		 *)
                                                                   	
	MesAuxHtOpenSectLine225kV					: BOOL;		       	(* AuxHtOpenSectLine225kV*)
	MesAuxHtCloseSectLine225kV					: BOOL;		       	(* AuxHtCloseSectLine225kV*)
                                                                   	
	                                                               	
	MesAuxHtOpenSectMalt						: BOOL;		       	(* AuxHtOpenSectMalt*)
	MesAuxHtCloseSectMalt						: BOOL;		       	(* AuxHtCloseSectMalt*)
                                                                   	
	MesAuxHtTeleCondamnSl225kV				 	: BOOL;		       	(* AuxHtTeleCondamnSl225kV			*)
	MesAuxHtDeTeleCondamnSl225kV				: BOOL;            	(* AuxHtDeTeleCondamnSl225kV		*)
	MesAuxHtTelecommandeRelestActif				: BOOL;		       	(* AuxHtTelecommandeRelestActif		*)
	MesAuxHtTelecommandeRelestPassif			: BOOL;	           	(* AuxHtTelecommandeRelestPassif	*)
	                                                               
	// Door Sensor, Fire Alarm, Local/Remote, Emergency Stop	   
	                                                            
	MesLocalRemoteOperation                  	: BOOL;            	(*LocalRemoteOperation    *)


	MesAlarmCom									: BOOL ; 		   	(* Communication Error with I35 module *) 
	MesCP_Read									: BOOL ;  			(* Cal : Read function enable *)

	MesAlarmCode1								: WORD ; 			(* Internal Akuo Alarm Code   *)
	MesAlarmCode2								: WORD ; 			(* Internal Akuo Alarm Code   *)
	MesAlarmCode3								: WORD ; 			(* Internal Akuo Alarm Code   *)
	MesWarningCode1								: WORD ; 			(* Internal Akuo Warning Code *)
	MesWarningCode2								: WORD ; 			(* Internal Akuo Warning Code *)  
	MesWarningCode3								: WORD ; 			(* Internal Akuo Warning Code *)
	MesWarningCode4								: WORD ; 			(* Internal Akuo Warning Code *)  
	MesWarningCode5								: WORD ; 			(* Internal Akuo Warning Code *) 
    MesWarningCode6								: WORD ; 			(* Internal Akuo Warning Code *)     
	MesEventCode1								: WORD ; 			(* Internal Akuo Event Code   *)  
	MesEventCode2								: WORD ; 			(* Internal Akuo Event Code   *) 
	MesEventCode3								: WORD ; 			(* Internal Akuo Event Code   *)  			                                                   			                                               
	
END_STRUCT
END_TYPE

// ---- 01_Equipement_Library/PCS/PCS.TcDUT
///////////
// Structure for CtrlPcs Jema .  
//////////
TYPE PCS :
STRUCT
// PCS Controller  Measures
	MesP 						: REAL;  		// (kW)  Active Power 
	MesQ 						: REAL;  		// (kVAr) Reactive Power
	MesPdc 						: REAL;  		// (kW)  DC Power 
	MesCosPhi 					: REAL;  		// (p.u) Power factor
	MesU 						: REAL;  		// (V) 	AC Voltage measure
	MesFreq						: REAL;			// (Hz) Main Bus Freq
	MesUdc 						: REAL;  		// (V) 	DC Voltage measure
	MesI 						: REAL; 		// (A) 	Total AC current 
	MesIdc 						: REAL; 		// (A) 	Total DC current from batteries (+ = discharge)
	MesState					: WORD;			// (NA) [P,H,B] Bit0: 1 = Not Available (AC or DC breaker open or AllAcContactorsOpened), Bit1: GridMode: 1=grid
	MesTemp						: REAL;			// (°C) Temperature sensor
	MesHumidity					: REAL;			// (%) Humidity sensor
	MesPrecharge				: BOOL;			// (NA) Precharge indicator      
	MesDcBreaker				: BOOL;			// (NA) Dc Breaker status      
	MesSoCLimitReached			: BOOL; 		// (NA) SoC limit reached
    MesAcBreaker				: BOOL; 		// (NA) Ac Breaker status
	MesHeartBeat				: WORD; 		// (NA) HeartBeat of the Inverter
	MesS_BatChargeMax			: REAL;			// (kVA) Max apparent power available for Charge based on load factor
	MesS_BatDischargeMax		: REAL;			// (kVA) Max apparent power available for discharge based on load factor
	MesNbPcsConnected			: UINT; 		// (NA) Number of online PCS 
	MesAtLeastOnePcsConnected	: BOOL; 		// (NA) At least one Pcs connected and not in alarm
	MesOpeFlag					: WORD;			// (NA) Operation flag from PCS
	MesWarning 					: BOOL; 		// (NA) PCS Controller general Warning 
	MesComAlarm					: BOOL; 		// (NA) PCS Controller Communication fault
	MesComWarning				: BOOL;			// (NA) PCS Controller Communication warning
	MesOnGrid 					: BOOL; 		// TRUE if AFE in ONgrid Mode.
	MesOffGrid 					: BOOL; 		// TRUE if AFE in Offgrid Mode.                 	
	MesFreqReg_Active			: BOOL; 		// (NA) Is the frequency regulation active : True = FreqReg Active
	MesUReg_Active				: BOOL; 		// (NA) Is the voltage regulation active : True = UReg Active
	MesSnom						: REAL; 		// (kW) Nominal power read on Controller
	MesAvailability				: REAL; 		// (%) Availability of the inverter
	MesAlarmCode				: WORD;			// (NA) Internal Akuo AlarmCode
	MesWarningCode				: WORD; 		// (NA) Internal Akuo WarningCode
	MesEventCode				: WORD;			// (NA) Internal Akuo EventCode
	OUT_CmdStop					: BOOL; 		// (NA) Stop  sent to the Controller
	OUT_CmdStart				: BOOL;			// (NA) Start sent to the Controller
	OUT_CmdStandby				: BOOL;			// (NA) Soft stop sent to the Controller
	OUT_CmdInvLocal				: BOOL;			// (NA) If true, INV is excluded from regulation
	OUT_CmdP					: BOOL;			// (NA) P setpoint is enabled
	OUT_CmdQ					: BOOL;			// (NA) Q setpoint is enabled
	OUT_CmdCosPhi				: BOOL;			// (NA) CosPhi setpoint is enabled
	OUT_CmdBlackStart			: BOOL;			// (NA) Blackstart order sent to the controller
	OUT_CmdFreqregMode			: BOOL;			// (NA) Frequency regulation mode sent to the controller
	OUT_CmdUregMode				: BOOL;			// (NA) Voltage regulation mode sent to the controller
	OUT_CmdMicroCyclingMode		: BOOL;			// (NA) MicroCycling is active
	OUT_CmdGridMode				: BOOL;			// (NA) Mode of the PCS :  FALSE = Grid Feeder, TRUE = Grid Former
	OUT_CmdOpenAc				: BOOL;			// (NA) Open AC breaker order sent to controller
	OUT_CmdOpenDc				: BOOL;			// (NA) Open DC breaker order sent to controller
	OUT_SetptP					: REAL; 		// (kW) Active power setpoint 
	OUT_SetptSMax				: REAL;			// (kVA) Upper range of the Apparent Power setpoint
	OUT_SetptPMax				: REAL;			// (kW) Upper range of the Active Power setpoint
	OUT_SetptPMin				: REAL;			// (kW) Lower range of the Active Power setpoint
	OUT_SetptQ					: REAL; 		// (kVAr) Reactive power setpoint 
	OUT_SetptQMax				: REAL;			// (kVAr) Upper range of the Reactive Power setpoint
	OUT_SetptQMin				: REAL;			// (kVAr) Lower range of the Reactive Power setpoint
	OUT_SetptCosPhi				: REAL;			// (NA) CosPhi setpoint
	OUT_MesV					: REAL;			// (V) Measure of the voltage sent to the Inverter for its regulation
	OUT_SetptV					: REAL;			// (V) Setpoint of the voltage sent to the Inverter for the OffGrid Mode
	OUT_SetptF					: REAL;			// (Hz) Setpoint of the frequency sent to the Inverter for the OffGrid Mode

	MesCP_Read					: BOOL := TRUE;	// (NA) CP to read values from PCS
	MesCP_Write					: BOOL := TRUE;	// (NA) CP to write values from PCS
	
END_STRUCT
END_TYPE

// ---- 01_Equipement_Library/PCS/PCS_Jema.TcDUT
///////////
// Structure for CtrlPcs Jema .  
//////////
TYPE PCS_Jema :
STRUCT
// PCS Controller  Measures
	AX_PowerCol					: ARRAY[1..3] OF PowerCol;

	MesData						: PCS ; 
	
END_STRUCT
END_TYPE

// ---- 01_Equipement_Library/PCS/PCS_PE.TcDUT
///////////
// Structure for CtrlPcs Jema .  
//////////
TYPE PCS_PE :
STRUCT
// PCS Controller  Measures
	AX_PowerCol					: ARRAY[1..6] OF PowerCol_PE;		(* PE Module*)
	
	MesData						: PCS ; (* MesData*)
	
	MesP_ChargeMax				: REAL ;		(* (%)	Max active power setpoint. SV4.2.1a	*)
	MesP_DischargeMax			: REAL ;		(* (%)	Max active power setpoint. SV4.2.1b	*)
	
	//Electrical Measurements	
	MesI1						: REAL; (* (A) Current phase 1 (R). INV: SV1.4 Grid current I1 (HEMK)															*)
	MesI2						: REAL; (* (A) Current phase 2 (S). INV: SV1.5 Grid current I2 (HEMK)															*)
	MesI3						: REAL; (* (A) Current phase 3 (T). INV: SV1.6 Grid current I3  (HEMK)															*)
	MesU12						: REAL; (* (V) Phase AB RMS voltage (line to line)at grid side of AC circuit breaker CB501. INV: SV1.1 Grid voltage RS (HEMK)	*)
	MesU23						: REAL; (* (V) Phase BC RMS voltage (line to line)at grid side of AC circuit breaker CB501. INV: SV1.2 Grid voltage ST(HEMK)	*)
	MesU31						: REAL; (* (V) Phase CA RMS voltage (line to line)at grid side of AC circuit breaker CB501. INV: SV1.3 Grid voltage TR (HEMK)	*)

	MesHumidity					: REAL;			(* (%) Humidity sensor	*)
	MesPconnected				: REAL; (* (%) Current available active power. INV: SV4.1.2 P limit inst 														*)  
	MesQconnected				: REAL; (* (%) Current available reactive power. INV: SV4.2.2 Q limit inst 														*)                                                      									

	MesIDState_InsuResistor_DC	: WORD ; (* (NA) Status of insulation protection. 0 = Idle, 1= Inter measurement quard, 2=measurement in progress, 3=self-test in progress, 4=risk addressed state SV3.1.1 *)
	MesInsuResistor_AC			: REAL;	(* (Ohms) AC Insulation Resistance. INV: SV3.2.2  Resistor 																*)
	MesIDState_InsuResistor_AC	: WORD ; (* (NA) Status of insulation protection. 0 = Idle, 1= Inter measurement quard, 2=measurement in progress, 3=self-test in progress, 4=risk addressed state SV3.1.1 *)
	MesInsuResistor_DC			: REAL;	(* (Ohms) DC Insulation Resistance. INV: SV3.2.1  Resistor 		*)

	MesUdc_Input1		 		: REAL ; (* (V) DC Voltage Bus 1 . INV : SV2.1.1 *)
	MesUdc_Input2		 		: REAL ; (* (V) DC Voltage Bus 2 . INV : SV2.1.2*)
	MesUdc_Input3		 		: REAL ; (* (V) DC Voltage Bus 3 . INV : SV2.1.3*)
	MesUdc_Bat1		 			: REAL ; 	(* (V) DC Voltage BESS 1 . INV : SV2.4.1*)
	MesUdc_Bat2		 			: REAL ; 	(* (V) DC Voltage BESS 2 . INV : SV2.4.2*)
	MesUdc_Bat3		 			: REAL ; 	(* (V) DC Voltage BESS 3 . INV : SV2.4.3*)
	MesPdc_Input1		 		: REAL ; (* (V) DC Power Bus 1 . INV : SV2.5a*)
	MesPdc_Input2		 		: REAL ; (* (V) DC Power Bus 2 . INV : SV2.5b*)
	MesPdc_Input3		 		: REAL ; (* (V) DC Power Bus 3 . INV : SV2.5c*)
	MesIdc_RFI_Input1    		: REAL ; (* (V) RFI Current  Bus 1 . INV : SV2.11a*)
	MesIdc_RFI_Input2    		: REAL ; (* (V) RFI Current  Bus 2 . INV : SV2.11b*)
	MesIdc_RFI_Input3	 		: REAL ; (* (V) RFI Current  Bus 3 . INV : SV2.11c*)
	MesIdc_Input1				: REAL; (*(A) SV2.6a DC input current*)
	MesIdc_Input2				: REAL; (*(A) SV2.6b DC input current*)
	MesIdc_Input3				: REAL; (*(A) SV2.6c DC input current*)

	//Status Summary
	MesIDState					: UINT; (* (NA) Current inverter status . INV : SV4.1.3                                                    *)                 	
	MesAlarmID					: WORD;	(* (NA) Alarm ID of the currently active event.  INV : SV4.1.1    *)
	MesWarningID				: WORD;	(* (NA) Warning ID of the currently active event.  INV : SV4.1.2    *)
	MesEventID					: WORD;	(* (NA) Event ID of the currently active event.  INV : SV9.1.1 :Last Event    *)
                    	
	// Inverter's Control Cabinet  Status                                                                       											
	MesTemp_IGBTmax				: REAL; 		 (* (C) Maximum IGBT temperature. INV: SV4.1.5 Max IGBTs temperature											*)
	MesTemp_PowerColmax			: REAL; 		 (* (C) Maximum power column temperature. INV: SV4.1.6 Max modules temperature									*)
 
	MesReadModule				: UINT;		(* (NA) module read *)
	MesIDState_PowerCol			: WORD ; 	(* (NA) Running modules (0 = stopped, 1 =running). Module 1 is the first from the right. SV9.1.1															*)
               	                                                   	                                						
	// Reset command        	                                                                     	                                						
	OUT_CmdReset 				: BOOL; 		 (* (NA) OUT reset command. INV: Reset command 43012															*)
	MesCalibrationState		 	: WORD;			(*(NA) it's a state to know if the calibration is ongoing or not, (0=running, 1=Discharging the batteries started, 2=20min hold finished, starting to send setpt of 0 for 20min, 3=Charging started*)
	MesBMSSelected				: WORD;
	OUT_SetptPMax_IMDicharge1	: REAL;
	OUT_SetptPMax_IMDicharge2	: REAL;
	OUT_SetptPMax_IMCharge1		: REAL;
	OUT_SetptPMax_IMCharge2		: REAL;
	MesSelector 				: BOOL;
	
	
END_STRUCT
END_TYPE

// ---- 01_Equipement_Library/PCS/PowerCol_JemaAlarms.TcDUT
TYPE PowerCol_JemaAlarms :
STRUCT

// ALARM0 bAlarm1
		MesI1_Alm			: BOOL; 	//RegAlarms0: I1_Alm
		MesI2_Alm			: BOOL; 	//RegAlarms0: I2_Alm
		MesI3_Alm			: BOOL; 	//RegAlarms0: I3_Alm
		MesVdc_High_Alm		: BOOL; 	//RegAlarms0: Vdc_High_Alm
		MesVdc_Low_Alm		: BOOL; 	//RegAlarms0: Vdc_Low_Alm
		                            	// 
		MesU12_High_Alm		: BOOL; 	//RegAlarms0: U12_High_Alm
		MesU12_Low_Alm		: BOOL; 	//RegAlarms0: U12_Low_Alm
		MesU23_High_Alm		: BOOL; 	//RegAlarms0: U23_High_Alm
		MesU23_Low_Alm		: BOOL; 	//RegAlarms0: U23_Low_Alm
		MesU31_High_Alm		: BOOL; 	//RegAlarms0: U31_High_Alm
		MesU31_Low_Alm		: BOOL; 	//RegAlarms0: U31_Low_Alm
		MesVd_High_Alm		: BOOL; 	//RegAlarms0: Vd_High_Alm
		MesVd_Low_Alm		: BOOL; 	//RegAlarms0: Vd_Low_Alm
		MesVdc_Neg			: BOOL; 	//RegAlarms0: Vdc_Neg
		                            	//   :blabla
										//wAlarmCode
		
// ALARM1 bAlarm1
		MesU1223_Unbalance	: BOOL;		//RegAlarms1: U1223_Unbalance
		MesU2331_Unbalance	: BOOL;		//RegAlarms1: U2331_Unbalance
		MesU3112_Unbalance	: BOOL;		//RegAlarms1: U3112_Unbalance
		MesInvertedPhase	: BOOL;		//RegAlarms1: InvertedPhase
		MesI12_Unbalance	: BOOL;		//RegAlarms1: I12_Unbalance
		MesI23_Unbalance	: BOOL;		//RegAlarms1: I23_Unbalance
		MesI31_Unbalance	: BOOL;		//RegAlarms1: I31_Unbalance
		MesCouplingTimeout	: BOOL;		//RegAlarms1: CouplingTimeout
		MesF_High			: BOOL;		//RegAlarms1: F_High
		MesF_Low			: BOOL;		//RegAlarms1: F_Low
		MesGrndFault		: BOOL;		//RegAlarms1: GrndFault
		MesVaristor			: BOOL;		//RegAlarms1: Varistor
		MesPcbOverTemp		: BOOL;		//RegAlarms1: PcbOverTemp
		MesHeatsinkOverTemp	: BOOL;		//RegAlarms1: HeatsinkOverTemp
		                           		// 
		MesOvertempHyst		: BOOL;		//RegAlarms1: OvertempHyst
		//wAlarmCode
// ALARM2 bAlarm1
										// 
                                    	// 
                                    	// 
                                    	// 
		MesGridCbOpened		: BOOL;		//RegAlarms2: GridCbOpened
		MesGridCbTrip		: BOOL;		//RegAlarms2: GridCbTrip
										//
		                           		// 
		MesGridContactFail	: BOOL;		//RegAlarms2: GridContactFail 
		MesDoorOpened		: BOOL;		//RegAlarms2: DoorOpened 
		                           		// 
		                           		// 
		MesVdcPrechargewrong: BOOL;		//RegAlarms2: VdcPrechargewrong 
		                           		// 
		MesOverVoltHyst		: BOOL;		//RegAlarms2: OverVoltHyst 
		MesIdcMax			: BOOL;		//RegAlarms2: IdcMax 
		//wAlarmCode
		
//ALARM3   bAlarm1                         
		MesSKIIP1			: BOOL; 	//RegAlarms3: SKIIP1
		MesSKIIP2			: BOOL; 	//RegAlarms3: SKIIP2
		MesSKIIP3			: BOOL; 	//RegAlarms3: SKIIP3
		MesSKIIP_OT			: BOOL; 	//RegAlarms3: SIIP_OT
		MesFPGA_WdogTrip	: BOOL; 	//RegAlarms3: FPGA_WdogTrip
		MesStopEverything	: BOOL; 	//RegAlarms3: StopEverything
		MesIMax				: BOOL; 	//RegAlarms3: IMax
		MesEmergencyStop	: BOOL; 	//RegAlarms3: EmergencyStop
		MesImdWarning		: BOOL; 	//RegAlarms3: ImdWarning
		MesImdFault			: BOOL; 	//RegAlarms3: ImdFault
		                            	//RegAlarms3:  
		MesCoilOverTemp		: BOOL; 	//RegAlarms3: CoilOverTemp
		                            	//RegAlarms3:  
		MesAlrmGrp1_Curr	: BOOL; 	//RegAlarms3: AlrmGrp1_Curr
		MesAlrmGrp2_Curr	: BOOL; 	//RegAlarms3: AlrmGrp2_Curr
		MesShortCircuit_DC	: BOOL; 	//RegAlarms3: ShortCircuit_DC
		//wAlarmCode
// ALARM4 bAlarm1
		MesBatError			: BOOL;		//RegAlarms4: BatError
		MesBatCtlStop		: BOOL;		//RegAlarms4: BatCtlStop
		MesBatComErrors		: BOOL;		//RegAlarms4: BatComErrors
		MesPowerUnbalance	: BOOL;		//RegAlarms4: PowerUnbalance
		MesOverpower		: BOOL;		//RegAlarms4: Overpower
		//wAlarmCode
		
END_STRUCT
END_TYPE

// ---- 01_Equipement_Library/PCS/PowerCol.TcDUT
///////////
// Structure For Jema Module 
//////////
TYPE PowerCol :
STRUCT
		MesP 						: REAL; 		// {1}(kW) Active Power output (AC) of PCS
		MesQ 						: REAL; 		// {1}(kVAr) Reactive AC Power Produced by PCS 
		MesPdc						: REAL ; 		// {1}(kW) DC Power . 
		MesCosPhi 					: REAL;  		// {0}(p.u) Power factor
		MesFreq						: REAL ; 		// {0}(Hz) Frequency
		MesTemp						: REAL ; 		// {0}(°C) PCS Internal Temperature
		MesU 						: REAL;  		// {0}(V) AC Voltage measure
		MesUdc 						: REAL;  		// {0}(V) DC Voltage measure
		MesI 						: REAL; 		// {0}(A) Total AC current 
		MesI1						: REAL ; 		// {0}(A) Phase 1 AC Current
		MesI2						: REAL ;        // {0}(A) Phase 2 AC Current
		MesI3						: REAL ;        // {0}(A) Phase 3 AC Current
		MesIdc 						: REAL; 		// {0}(A) Total DC current from batteries (+ = discharge)
		MesPavailable 				: REAL;  		// {1}(kW) Available PCS Power 
		MesPconnected				: REAL ; 		// {0}(kW) Connected PCS Power 
		MesDcSwitchClosed			: BOOL ; 		// {0}(NA) Position of the DC Switch : True = Switch closed
		MesAcSwitchClosed			: BOOL ; 		// {0}(NA) Position of the AC Switch : True = Switch closed
		MesTempControl      		: REAL ; 		// {0}(°C) Temperature of control card
		MesTempPowerUnit    		: REAL ;		// {0}(°C) Temperature of Power Unit
		MesTempCabinet      		: REAL ; 		// {0}(°C) Cabinet temperature
		MesTempCoil1        		: REAL ; 		// {0}(°C) Coil temperature
		MesRegAlarm0        		: WORD ; 		// {0}Alarm Word of PCS
		MesRegAlarm1        		: WORD ; 		// {0}Alarm Word of PCS 
		MesRegAlarm2        		: WORD ; 		// {0}Alarm Word of PCS 
		MesRegAlarm3        		: WORD ;  		// {0}Alarm Word of PCS
		MesRegAlarm4        		: WORD ;  		// {0}Alarm Word of PCS
		MesDeratingWord				: WORD ;		// {0}Derating word of PCS
		MesHeartbit					: REAL ;		// {0}Heartbit
		MesDoorOpened				: BOOL ;		// {1}Door of the Power module is opened	
		
		MesJemaAlarms				: PowerCol_JemaAlarms;

			

END_STRUCT
END_TYPE

// ---- 01_Equipement_Library/PCS/PowerCol_PE.TcDUT
///////////
// Structure For Jema Module 
//////////
TYPE PowerCol_PE :
STRUCT
		
		MesData					: PowerCol ; (* MesData *) 

		AX_DCInputs			: ARRAY[1..10] OF  DCInputs_PE ;(* Object *) 
		
		MesIDState			: DWORD ;		(* (NA) 	Module status (SV9.3 PE documentation p.97)																*)
		MesTempmax			: REAL ;		(* (C) 		Maximum IGBT temperature of the selected module															*)
		MesStateIO			: WORD ;		(* (NA) 	0: Open, 1: Closed. Bit 1 =  fan contactor, Bit 2 = main AC contactor, Bit 3 = AC soft charge contactor, Bit 4 = LCL filter contactor, Bit 5 = DC contactor , Bit 6 = reserved, Bit 7 = if open : overheating in the coil, Bit 8 = fan contactor feedback, Bit 9 = AC main contactor feedback, Bit 10 = AC soft charge contactor feedback, Bit 11 = LCL filter contactor feedback , Bit 12 = DC contactor feedback *) 		
		MesHygro			: REAL ; 		(* (%) 		Percentage of humidity																					*)
		MesAlarmID			: BYTE ; 		(* (NA)  PowerColumn Alarm ID  . W65 to W116  *)
			

END_STRUCT
END_TYPE

// ---- 01_Equipement_Library/ProtectRelay/ProtectRelay.TcDUT
///////////
// Structure For I35. Main Operating Data to be saved (ex: OPC).  
//////////
TYPE ProtectRelay :
STRUCT
		MesI1						: REAL ; 			(* (A) Maximal Current measured before fault on phase 1*)
		MesI2						: REAL ;			(* (A) Maximal Current measured before fault on phase 2*)
		MesI3						: REAL ;			(* (A) Maximal Current measured before fault on phase 3*)
		MesI0						: REAL ; 			(*(A) Measured  maximal residual current               *)
		MesI						: REAL ;			(*(A) Phase current value (averaged)               	   *)
		                                        		                                                    
		MesFreq						: REAL ;			(* (Hz) Frequency measured                             *)
		                                        		                                                    
		MesImax1					: REAL ; 			(* (A) AC Max current during Fault phase 1             *)
		MesImax2                    : REAL ; 			(* (A) AC Max current during Fault phase 2             *)
		MesImax3                    : REAL ; 			(* (A) AC Max current during Fault phase 3		       *)
		MesImax0                    : REAL ; 			(* (A) AC Max residual current during Fault	           *)
		
		MesTripped                  : BOOL ;            (* Trip Synthesis *)                                        		                                                    
		MesAlarmCom					: BOOL ;			(* Communication Error with Sepam                      *)
                                                		                                                   
		MesAlarmTCS					: BOOL ; 			(* TCS in fault. RPN can not trip anymore              *)
		MesAlarmImax				: BOOL ; 			(* Imax alarm, ANSI Trip 50, 51 , 50G, 51G Synthesis                                       *)
		MesAlarmUmin				: BOOL ;			(* Short GTE Fault                                     *)
		MesAlarmUmin_Long			: BOOL ;			(* Long GTE FAULT                                      *)
      	MesAlarm_GTE3Time			: BOOL ; ;			(* 3 GTE FAULT   in 30 minutes                                   *)
		MesU12                      : REAL ;            (* (V) Voltage between phase 2 and phase 1 *)
		MesU23                      : REAL ;            (* (V) Voltage between phase 3 and phase 2 *)     
		MesU31                      : REAL ;            (* (V) Voltage between phase 1 and phase 3 *)                                                                                              
		
		MesAlarmWatchdog	       	: BOOL ;            (* (nA) Watchdog *) 

		MesCP_Read					: BOOL := FALSE;	(* Cal Read function enable                            *)
		MesCP_Write					: BOOL := FALSE;	(* Cal Write function enable                           *)
		                                                                                                     
		MesAlarmCode				: WORD ; 			(* (NA) Internal Akuo AlarmCode                        *)
		MesWarningCode				: WORD ; 			(* (NA) Internal Akuo WarningCode                      *)
		MesEventCode				: WORD ; 			(* (NA) Internal Akuo EventCode		                   *)
		
END_STRUCT
END_TYPE

// ---- 01_Equipement_Library/ProtectRelay/ProtectRelay_S48.TcDUT
///////////
// Structure For I35. Main Operating Data to be saved ( ex: OPC ) .  
//////////
TYPE ProtectRelay_S48 :
STRUCT
	
		MesData						: ProtectRelay;			(*	(NA) Protection relay									    *)
                                                        	                                               
		                                    				                                                             
		MesU						: REAL;					(* (V) Average Phase to Phase Voltage                           *)
	                                                    	
		MesV1						: REAL ;        		(* (V) Average Phase to Phase Voltage                           *)
		MesV2						: REAL ;				(* (V) Average Phase to Phase Voltage                           *)
		MesV3						: REAL ;				(* (V) Average Phase to Phase Voltage                           *)
       			                                        	                   
		MesP						: REAL; 				(* (Kw)Power on Grid                                            *)
		MesQ						: REAL;					(* (kvar) Power on grid                                         *)
		MesS						: REAL;					(* (KVA) Power apparent                                         *)
		MesCosPhi					: REAL;					(* (NA) power factor                                            *)
		MesTanPhi					: REAL; 				(* (NA) Cal : tan Phi                                           *)
		   

                                 			                                                        
		MesStopPP_UminLong			: BOOL; 				(* (NA) PP is stopping during 2min, because of Long GTE fault	*)
		                                    			                                                          
		EActProd					: REAL; 				(* (MWh) Active Energy Produced                                 *)
		EActCons					: REAL; 				(* (MWh) Active Energy Consummed                                *)
		EReactProd					: REAL; 				(* (MVArh) Reactive Energy Produced                             *)
		EReactCons					: REAL; 				(* (MVArh) Reactive Energy Consummed                            *)
		                                    			                                                           
	// Relais Input                         			
		Input11						: BOOL;					(* (NA) Input 11 du relais de protection                        *)
		Input12                     : BOOL;					(* (NA) Input 12 du relais de protection                        *)
		Input13                     : BOOL;					(* (NA) Input 13 du relais de protection                        *)
		Input14                     : BOOL;					(* (NA) Input 14 du relais de protection                        *)
		Input21						: BOOL;					(* (NA) Input 21 du relais de protection                        *)
		Input22						: BOOL;					(* (NA) Input 22 du relais de protection                        *)
		Input23						: BOOL;					(* (NA) Input 23 du relais de protection                        *)
		Input24						: BOOL;					(* (NA) Input 24 du relais de protection                        *)
		Input25						: BOOL;					(* (NA) Input 25 du relais de protection                        *)
		Input26						: BOOL;					(* (NA) Input 26 du relais de protection                        *)
		
				
END_STRUCT
END_TYPE

// ---- 01_Equipement_Library/Router/Router.TcDUT
TYPE Router :
STRUCT
		MesWatchdog	        : BOOL ; 	(* Watchdog*)
		
		MesAlarmCode		: WORD ;	(* (NA) Internal Akuo AlarmCode		*)
		MesWarningCode		: WORD ; 	(* (NA) Internal Akuo WarningCode   *)
		MesEventCode		: WORD ; 	(* (NA) Internal Akuo EventCode	    *)
		
END_STRUCT
END_TYPE

// ---- 01_Equipement_Library/Router/Router_Standard.TcDUT
TYPE Router_Standard :
STRUCT
		MesData				: Router ;  (* Object *)

		
END_STRUCT
END_TYPE

// ---- 01_Equipement_Library/Sensors/ANA/ANA_Standard.TcDUT
TYPE ANA_Standard :
STRUCT
	MesData : ANA; (* Child structure*)

END_STRUCT
END_TYPE

// ---- 01_Equipement_Library/Sensors/ANA/ANA.TcDUT
TYPE ANA :
STRUCT
	Value 					: REAL ;	(* (-) Analogic Value 					*)
	                                    
	MesAlarmCode			: WORD ;	(* (NA) Internal Akuo AlarmCode     *)
	MesWarningCode			: WORD ;    (* (NA) Internal Akuo WarningCode   *)
	MesEventCode			: WORD ;    (* (NA) Internal Akuo EventCode		*)

END_STRUCT
END_TYPE

// ---- 01_Equipement_Library/Sensors/COM/AllInOne.TcDUT
TYPE AllInOne :
STRUCT
	
	MesWindSp 			: REAL ;		(* (m/s)	 Wind speed measurement of the weather station												        *)
	MesWindDir 			: REAL ;		(* (°) 		 Wind direction measurement of the weather station                                                  *)
	MesHygro			: REAL ;		(* (%) 		 Humidity measurement of the weather station                                                        *)
	MesTemp_Amb 			: REAL ;		(* (°C)		 Ambiant temperature measurement of the weather station                                             *)
	MesDewPoint			: REAL ;		(* (%) 		 Dew point measure of weather station                                                               *)
	MesRain1			: REAL ;		(* (count/h) Rain rate                                                                                          *)
	MesRain2			: REAL ;		(* (count/h) Rain rate                                                                                          *)
	MesRain3			: REAL ;		(* (count/h) Rain rate                                                                                          *)
                                        (*                                                                                                              *)
	MesAlarmWindSp		: REAL ;		(* Alarm for the Wind speed : 0=OFF, 1 = Lower threshold, 2 = Higher threshold                                  *)
	MesAlarmWindDir		: REAL ;		(* Alarm for the Wind direction : 0=OFF, 1 = Lower threshold, 2 = Higher threshold                              *)
	MesAlarmTemp		: REAL ;		(* Alarm for the temp sensor : 0=OFF, 1 = Lower threshold, 2 = Higher threshold                                 *)
	MesAlarmHygro		: REAL ;		(* Alarm for the humidity sensor : 0=OFF, 1 = Lower threshold, 2 = Higher threshold                             *)
	MesAlarmDewPt		: REAL ;		(* Alarm for the dew point sensor : 0=OFF, 1 = Lower threshold, 2 = Higher threshold                            *)
	MesAlarmRain1		: REAL ;		(* Alarm for the rain sensor : 0=OFF, 1 = Lower threshold, 2 = Higher threshold                                 *)
	MesAlarmRain2		: REAL ;		(* Alarm for the rain sensor : 0=OFF, 1 = Lower threshold, 2 = Higher threshold                                 *)
	MesAlarmRain3		: REAL ;		(* Alarm for the rain sensor : 0=OFF, 1 = Lower threshold, 2 = Higher threshold                                 *)
	                                    (*                                                                                                              *)
	MesAlarmCode		: WORD ;  	    (*                                                                                                              *)
	MesWarningCode		: WORD ;  	    (*                                                                                                              *)
	MesEventCode		: WORD ; 	    (*                                                                                                              *)
	
END_STRUCT
END_TYPE

// ---- 01_Equipement_Library/Sensors/COM/SMP1X.TcDUT
TYPE SMP1X :
STRUCT
	MesData						: ANA; 			(**)

	
	MesAlarm					: REAL;			(**)
	MesCP_Read					: BOOL;			(**)

END_STRUCT
END_TYPE

// ---- 01_Equipement_Library/Sensors/TOR/TOR.TcDUT
TYPE TOR :
STRUCT
	
	MesAlarmState 		 		: BOOL  ;		(* TRUE = ALARM													*)
	MesCountAlarm				: UDINT ; 		(* Count the number of time the alarm has been triggered.       *)
                                                (*                                                              *)
	MesAlarmCode				: WORD ;		(* (NA) Internal Akuo AlarmCode                                 *)
	MesWarningCode				: WORD ;   	 	(* (NA) Internal Akuo WarningCode                               *)
	MesEventCode				: WORD ;	 	(* (NA) Internal Akuo EventCode		                            *)

END_STRUCT		
END_TYPE

// ---- 01_Equipement_Library/Sensors/TOR/TOR_Standard.TcDUT
TYPE TOR_Standard :
STRUCT
	
	MesData					: TOR ;		(* MesData 											 *)

END_STRUCT		
END_TYPE

// ---- 01_Equipement_Library/Transfo/Transfo.TcDUT
TYPE Transfo :
STRUCT
    MesWarningTemp				: BOOL ;	(* Transfo Temperature warning		    *)
    MesAlarmTemp				: BOOL ;	(* Transfo Temperature Alarm		    *)
    MesAlarmGas					: BOOL ;	(* Transfo Gas Alarm			        *)
    MesAlarmOilLevel			: BOOL ;	(* Transfo Oil Level Alarm		        *)
    MesAlarmsSynthesis			: BOOL ;	(* Transfo Synthesis Alarm              *)
                                                                             
	MesAlarmCode				: WORD ;  	(* (NA) Internal Akuo AlarmCode         *)
	MesWarningCode				: WORD ; 	(* (NA) Internal Akuo WarningCode       *)
	MesEventCode				: WORD ; 	(* (NA) Internal Akuo EventCode	        *)

END_STRUCT
END_TYPE

// ---- 01_Equipement_Library/Transfo/Transfo_MV.TcDUT
TYPE Transfo_MV :
STRUCT
	
	MesData						: Transfo ; (* MesData *)


END_STRUCT
END_TYPE

// ---- 01_Equipement_Library/UPS/UPS.TcDUT
///////////
// Structure for UPS. Main Operating Data to be saved (ex: OPC)  
//////////
TYPE UPS :
STRUCT
		MesDischarging				: BOOL ; 			(* (NA) Battery is discharging		*)
		MesAlarm_Ulow				: BOOL ; 			(* (NA) Battery is almost empty     *)
		MesAlarmState				: BOOL ; 			(* (NA) Fault on the charger        *)
		MesUdc  					: REAL ; 			(* (V) DC Load voltage              *)
       		
		
		MesAlarmCode				: WORD ; 			(* Internal Akuo Alarm Code         *)
		MesWarningCode				: WORD ; 			(* Internal Akuo Warning Code       *)
		MesEventCode				: WORD ; 			(* Internal Akuo Warning Code 	    *)
        
		MesCP_Read					: BOOL := FALSE ;   (* Read function enable             *)
		MesAlarmCom					: BOOL ; 			(* Communication alarm              *)
	
END_STRUCT
END_TYPE

// ---- 01_Equipement_Library/UPS/UPS_Eneris.TcDUT
///////////
// Structure For I35. Main Operating Data to be saved (ex: OPC).  
//////////
TYPE UPS_Eneris :
STRUCT
	// I35 Data measures
		MesData                     : UPS;  (* MesData *)
		
END_STRUCT
END_TYPE

// ---- 04_Application/IO/ST_AI.TcDUT
TYPE ST_AI :
STRUCT
		Value		  AT %I*	: INT	;
		Description 			: STRING	;

END_STRUCT
END_TYPE

// ---- 04_Application/IO/ST_AO.TcDUT
TYPE ST_AO :
STRUCT
		Value		  AT %Q*	: INT	;
		Description 			: STRING	;

END_STRUCT
END_TYPE

// ---- 04_Application/IO/ST_DI.TcDUT
TYPE ST_DI :
STRUCT
		Value		  AT %I*	: BOOL	;
		Description 			: STRING	;

END_STRUCT
END_TYPE

// ---- 04_Application/IO/ST_DO.TcDUT
TYPE ST_DO :
STRUCT
		Value		  AT %Q*	: BOOL	;
		Description 			: STRING	;

END_STRUCT
END_TYPE

// ---- 04_Application/OPC/AllDataR.TcDUT
TYPE AllDataR :
	
// 	REGLES : 														
// 	Mettre seulement les structures des produits 					
// 	Séparer les Structures (Pas AX_PTR mais PTR_1, PTR_2, ...)		
// 	Les noms des variables sont globales (Pas ION7650 mais PM) 		 
//	PP
//	PTR_1, PTR_2, PTR_3
//	INV		

STRUCT
	
//PP               	
	PP					: PP;              	   (* PP *)
	
//SUB_MV               	
	SUBMV				: SUBMV_Exd;       	   (* SUB.MV*)

// PTR        	
	PTR					: ARRAY[1..CstNbPTR_G] OF  PTR_Exd;        (* PTR *)

//WS                	
	WS					: WS_AGMA;              		(* WS *)
                                           		
//COM                                      		
	SMS					: ServerSms;       		(* SMS      *)
	MAIL				: ServerMail;      		(* MAIL     *)
	COM					: COM_Status;	   		(* COM      *)
	CSV					: ServerCSV;       		(* CSV      *)
	CSVData				: LoggerCSV;       		(* CSVData  *) 
	
//OPC
	MesAlarmCode		: WORD ; 				 (* OPC Alarm Code   *)
	MesWarningCode		: WORD ; 				 (* OPC Warning Code *)
	MesEventCode : ARRAY[1..9] OF WORD ; //Akuo EventCode
END_STRUCT

END_TYPE

// ---- 04_Application/OPC/AllDataWPulse.TcDUT

TYPE AllDataWPulse :
STRUCT
	//Communication
	CmdReset_ServerSMS			: BOOL;			(* Reset SMS Server *)
	CmdReset_ServerMail			: BOOL;			(* Reset Mail server *)
	CmdReset_Router_ADSL		: BOOL;			(* Restart ADSL router *)	
	CmdReset_Router_4G			: BOOL;			(* Restart 4G router *)
	CmdReset_IPC				: BOOL;			(* Restart IPC *)
	CmdDeleteAllSms				: BOOL;  		(* Delete all SMS in the buffer *)
	CmdChangeInfos_PhoneEmail	: BOOL;			(* Apply new changes in MAil and SMS infos *)
	CmdReadInfosFromTarget_PhoneEmail	: BOOL ; 	(* Get Saved configuration *)
	CmdTestSms					: BOOL;         (* Test SMS function *)
	
	
	CmdRestart_HH		      	: BOOL;			(* Restart HH *)
	CmdRestart_OPCUA 	   		: BOOL;			(* Restart OPCUA *)
	CmdRestart_OpenVPN 	 		: BOOL;			(* Restart OpenVPN *)
	CmdRestart_Teamviewer		: BOOL;			(* Restart Teamviewer *)
	CmdRestart_HMIServer 		: BOOL;			(* Restart HMIServer *)
	CmdRestart_Docker 	  		: BOOL;			(* Restart Docker *)	
	CmdRestart_Codesys 			: BOOL;			(* Restart Codesys *)	


	CmdRestart_PLC				: BOOL;			(* Restart PLC *)
	CmdForcedStay_Connect		: BOOL;			(* Force the power plant to remains connected during a code restart or reboot *)
	CmdIpLauncher				: BOOL;			(* Get the public IP of the power plant	*)                  
	CmdStart_Vpn				: BOOL;			(* Start VPN *)
	CmdStop_Vpn					: BOOL;			(* Stop VPN *)
                         
	// Maintenance and Test     
	CmdInhibAllWrite			: BOOL; 		(* Force all digital and analog output to FALSE when activated. Inhibate communication write *) 
	CmdAllowAllWrite			: BOOL; 		(* Force all digital and analog output to TRUE when activated.  Allow communication write *)
	CmdInhibAllRead				: BOOL; 		(* Force all digital and analog input to FALSE when activated. Inhibate communication read *)
	CmdAllowAllRead				: BOOL; 		(* Force all digital and analog input to FALSE when activated. Inhibate communication read  *)
	CmdWriteSetptTanPhi			: BOOL; 		(* PP Setpoint TanpHI *)
                           
	// SUB_MV                      
	CmdClose_MainMVCB			: BOOL; 		(* Close MainMVCB *)
	CmdOpen_MainMVCB			: BOOL;     	(* Open MainMVCB *)
	CmdReset_MainMVCB			: BOOL;     	(* Open MainMVCB *)	

	CmdOpen_FeederMVCB			: ARRAY[1..CstNbFeederMVCB_G] OF  BOOL;     (* Open FeederMVCB [ARRAY]*)
	CmdClose_FeederMVCB			: ARRAY[1..CstNbFeederMVCB_G] OF  BOOL;   	(* Close FeederMVCB [ARRAY]*)
	CmdReset_FeederMVCB			: ARRAY[1..CstNbFeederMVCB_G] OF  BOOL;   	(* Close FeederMVCB [ARRAY]*)
	                                        
	CmdStartLocalSetptP_PP		: BOOL;     	(*	Activate local setpoint at substation *)
	CmdStopLocalSetptP_PP		: BOOL;     	(*	Desactivate local setpoint at substation *)
	
	// PTR
	CmdOpen_PTR					: ARRAY[1..CstNbPTR_G] OF BOOL;		(*	Open corresponding PTR [ARRAY]*) 
	CmdClose_PTR				: ARRAY[1..CstNbPTR_G] OF BOOL;		(* Close corresponding PTR [ARRAY]*)
	
	// Inverter
	CmdStart_INV				: ARRAY[1..CstNbPTR_G] OF ARRAY[1..CstNbInv_PTR_G] OF BOOL;		(* Switch On inverter [ARRAY]*)
	CmdStop_INV					: ARRAY[1..CstNbPTR_G] OF ARRAY[1..CstNbInv_PTR_G] OF BOOL;     (* Switch Off inverter [ARRAY]*)
	CmdStartSetptP_INV			: ARRAY[1..CstNbPTR_G] OF ARRAY[1..CstNbInv_PTR_G] OF BOOL;     (* Activate local setpoint on inverter [ARRAY]*)
	CmdStopSetptP_INV			: ARRAY[1..CstNbPTR_G] OF ARRAY[1..CstNbInv_PTR_G] OF BOOL;		(* Desactivate local setpoint on inverter [ARRAY]*)
	CmdToggleCom_Read			: ARRAY[1..CstNbPTR_G] OF ARRAY[1..CstNbInv_PTR_G] OF BOOL;		(* Inverter Toggle Read Communcation [ARRAY]*) 
	CmdToggleCom_Write			: ARRAY[1..CstNbPTR_G] OF ARRAY[1..CstNbInv_PTR_G] OF BOOL;		(* Inverter Toggle Write Communcation [ARRAY]*)
	
	// UPS 
	CmdRestart_UPS48			: BOOL ; (*	Restart UPS *)
	
	
// GRID
	CmdAutCpl					: BOOL; 		(* Coupling authorization	*)
	CmdDisconnect				: BOOL; 		(* Powerplant disconnect order *)
	CmdEmergencyDisconnect		: BOOL; 		(* Powerplant Emergency disconnect order *)
	
	//Project specific ( France ) 
	CmdDisconnect_end			: BOOL; 		(* Powerplant disconnect order *)
	CmdEmergencyDisconnect_end	: BOOL; 		(* Powerplant Emergency disconnect order *)
	CmdStartPReg				: BOOL ; 		(* Activate P regulation from Grid   *)
	CmdStopPreg                 : BOOL ; 		(* Desactivate P regulation from Grid   *)
	CmdStartQReg                : BOOL ; 		(* Activate Q regulation from Grid   *)
	CmdStopQReg                 : BOOL ; 		(* Desactivate Q regulation from Grid   *)

           	
END_STRUCT
END_TYPE

// ---- 04_Application/OPC/AllValueW.TcDUT
TYPE AllValueW :
STRUCT
 // PP 
	SetptTanPhi_PP				: REAL; 										(* (p.u) TanPhi setpoint to regulate if the corresponding mode is activated *)

// SMS 	
	AX_NbPhone_OPC				: ARRAY[1..CstNbUser] OF STRING(26);			(* List of the phone number to be registered for SMS functions *)
	AX_SubscribedSms_OPC		: ARRAY[1..CstNbUser] OF BOOL;					(* List of subscription for SMS function *)
	AX_NamesUsers_OPC					: ARRAY[1..CstNbUser] OF STRING(50);	(* List of SMS user names *)
	AX_MailAddr_OPC				: ARRAY[1..CstNbUser] OF STRING(255);			(* Contient tous les numéros des utilisateurs *)
	AX_SubscribedMail_OPC		: ARRAY[1..CstNbUser] OF BOOL;					(* List of subscription fro MAIL function *)
	AX_UserLVL					: ARRAY[1..CstNbUser] OF WORD;					(* Bit-wise encoding of Alarm subscription (Check Config alarm document for bit signification) *)
	
// SUB	
	SetpP_SUB					: REAL;											(* (kW) Active Power setpoint to be regulated at Subatstion ( if local setpoint enabled) *)
    SetpQ_SUB					: REAL;											(* (kVAr) Reactive Power setpoint to be regulated at Subatstion ( if local setpoint enabled) *)
// PTR 
	SetpP_INV					: ARRAY[1..CstNbPTR_G] OF ARRAY[1..CstNbInv_PTR_G] OF  REAL;	(*(kW) Active Power setpoint to be regulated at the inverter ( if local setpoint enabled) *) 	
	
END_STRUCT
END_TYPE

// ---- 04_Application/CONFIG/GVL_BASE.TcGVL
///////////////////////
// DO NOT MODIFY :  
// Maximal number of objects  - Maximal array size 
////////////////////
VAR_GLOBAL CONSTANT 
	// PRODUCT 
	CstNbPTR_G					: BYTE := 4 ;  				// (NA) Number of PTR
	CstNbESS_G   				: BYTE := 3 ;  				// (NA) Number of ESS


	// EQUIPMENT
		//SUB_MV
	CstNbFeederMVCB_G			: BYTE	:= 3 ; 
		// PTR 
	CstNbInv_PTR_G				: BYTE := 2 ;				// Maximal Number of PV Inverters for PTR
	CstNbSB_INV_G				: BYTE := 32 ;				// Maximal Number of String box in inverter

		// EM 		
	CstNbEM_G					: BYTE := 1;				// Number of Energy Meters
		
		//ESS		
	CstNbPcs_ESS_G				: BYTE := 2  ;
	CstNbPowerCol_PCS_G			: BYTE := 3  ;				// Maximal Number of Power colonne by PCS
	CstNbHvac_ESS_G				: BYTE := 2  ;
	CstNbBAT_ESS_G				: BYTE := 2  ;
	CstNbRack_BAT_G				: BYTE := 2  ;
	CstNbModule_Rack_G			: BYTE := 25  ;
		
		//WS		
	CstNbPyrano					: UINT := 5;
	CstNbAnemo					: UINT := 1;
	CstNbPanTmp					: UINT := 4;
	CstNbAmbTmp					: UINT := 3;	
		
	// PP 
	CstNbCouplermax_G			: BYTE 	:= 100 ;			// Maximal number of ethercat devices 
	CstNbAlarmIO_G				: BYTE := 10 ; // Number of Event in PRG_IO.
	
	
	(*               SMS               							*)
	CstNbUser					: SINT:=10; //Nbr d'utilisateur utilisé par AX_Numtel
	CstNbCMD					: SINT:=20; //Nbr commande utilisé par AX_CMD_SMS
	CstNbAlarmCode				: INT:=213;  //Number of alarmcode use in AlarmManager
	
	// TIMEZONE
	    (* Indonesia East Standard Time Zone settings *)
        FRANCE_TZI : ST_TimeZoneInformation := (bias:=-60,
                                       		 				standardName:='Heure Française',
                                        					standardDate:=(wYear:=0,wMonth:=10,wDayOfWeek:=0,wDay:=27,wHour:=3),
                                        					standardBias:=0,
                                        					daylightName:='None',
                                        					daylightDate:=(wYear:=0,wMonth:=3,wDayOfWeek:=0,wDay:=31,wHour:=2),
                                        					daylightBias:=0);
			
		CstPhoneIndicator_G		: STRING := '+33';
			
			CstCycleTime_G		: INT := 10 ; 			// (ms) Cycle Time of the CPU FB Main 
			CstCycleTime_Annex	: INT := 100 ; 			// (ms) Cycle Time of the CPU FB Annex_Function

		CstNbRedundantVariableMax_G	: UINT := 553 ;
		CstNbParamOPCUA				: UINT := 100 ; 
	
END_VAR
VAR_GLOBAL
	sTimeGMT_G          	: STRING;				// Full Date Time for historization (GMT) 
	sTimeLocal_G		 	: STRING ;				// Local Time 
	CalGMTTimeStruct		: TIMESTRUCT ; 			// GMT Time Structure

	ParamOpenVpnFile		: STRING := '';			// Path to openvpn file. 
	ParamIpPublic 			: STRING(255);			// Public IP 
	MesSizeCdrive_PLC		: REAL := 100000 ; 		// (Mo) Remaining Disk space
	MesSizeCdrive_IndusPC	: REAL := 100000 ; 		// (Mo) Remaining Disk space
END_VAR

// ---- 04_Application/CONFIG/GVL_CFG.TcGVL
///////////////
// Configuration Files. Define Power Plant sizing and references. 
//////////////
VAR_GLOBAL 
		CstPLCBackup 			: BOOL := FALSE ;  			// TRUE if this PLC is used as a backup . 
		CstNetAmsId_Slave		: STRING(20):= '5.49.202.22.1.1'; //NetAMSId Slave .'5.79.170.90.1.1'
		CstNetAmsId_IndusPC		: STRING(20):= ''; // set '' if no Indus PLC
		//CstIPIEC104			: STRING := '10.101.111.1' ; 
		
		
END_VAR
	
VAR_GLOBAL 
	// Solar Classique //
		A1_PP					: FB_PP  ;  								// MCA Power Plant 
 
	// PRODUCT DEFINITION //
		//PTR 
		AX_PTR 					: ARRAY[1..CstNbPTR_G] OF FB_PTR ; 	 		// Array with AMG products
		
		//SUB_MV
		A1_SUBMV				: FB_SUBMV ;	 					 		// SUB_MV		
		
		//WEATHER STATION
		A1_WS					: FB_WS;
		
		//ESS 
		//AX_ESS				: ARRAY[1..CstNbESS_G] OF FB_ESS ; 
		
	// GLOBAL VARIABLE //
	
		CmdClearFault_G			: BOOL ; 									// (NA) Clear all permanent faults
		CmdInit_G				: BOOL ; 									// (NA) Global Init Action
		CstIPIEC104				: STRING := '10.111.109.1' ; 		
END_VAR

// ---- 04_Application/MAIN/MAIN.TcPOU
PROGRAM MAIN

VAR_INPUT PERSISTENT 
	ParamDisablePLCMaster			: BOOL ;  				(* If true  Force the Redundancy to be on the Slave PLC therefore, no read and write on FB and IO*)
	ParamForceRun					: BOOL ; 				(* Force the PLC to be in run mode .                                *)
	ParamInhibateGridLOC			: BOOL:= TRUE ;			(* Do not switch to slave PLC in case of GRID communication fault   *)
	ParamTest						: BOOL := TRUE ; 		(* If on , do not allow write commands at start up .                *)
	ParamStableOP					: TIME := T#5S ; 
END_VAR

VAR_OUTPUT
	OUT_CalRunningPLC_IO			: BOOL ; 
END_VAR

VAR

	// REDUNDANCY

		TON_Stable 				: TON ;
		FB_MasterBackup			: FB_HeartBeatMasterBackup ;  
 		PLC_ReadSymInfoByName1  : PLC_ReadSymInfoByName	;
		
		CalStableOp_G			: BOOL  ; 

		
	// DATETIME //	
		FB_LocalSystTime      	: FB_LOCALSYSTEMTIME;	// Get time function
		FB_ToGMT : FB_TzSpecificLocalTimeToSystemTime;	// Local to UTC Time function
		TON_Time				: TON;
		CalLocalTimeStruct_Temp: TIMESTRUCT;
		//init
		FB_GetSystemTime        : GETSYSTEMTIME;						// GEt time function
		
		FB_ToLocal 				: FB_FileTimeToTzSpecificLocalTime;		// UTC to local Time function
		fileTime        		: T_FILETIME;							// Filetime format for UTC Time 
		FileTimeLocal			: T_FILETIME;							// Filetime format for local time	

		
	//M_INIT VARIABLE //
		bInit					: BOOL := TRUE ;						// Initialization variable

	R_TRIG_Run: R_TRIG;
	F_TRIG_Run: F_TRIG;

END_VAR

// REDUNDANCY 
	// Heartbit Check
	// Check for ADS variable name every minute. 
	PLC_ReadSymInfoByName1(NETid := CstNetAmsId_Slave, Port:=851,Symname:='MAIN.FB_MasterBackup.nCounter', Start:= CalLocalTimeStruct.wSecond=0 OR bInit,TMOUT:= T#5S) ; 
	FB_MasterBAckup(sNetId:=GVL_CFG.CstNetAmsId_Slave, IdxGroup:=PLC_ReadSymInfoByName1.SYMINFO.idxGroup , IdxOff:=PLC_ReadSymInfoByName1.SYMINFO.idxOffset );

		FB_MasterBAckup.M_Backup() ; 
		FB_MasterBAckup.M_Master() ; 

// INITIALIZATION//
	IF bInit OR CmdInit_G THEN
		M_Init() ; 
		bInit := FALSE; 
	END_IF
	
//GLOBAL VARIABLE UPDATE //
// DateTime 
// Takes some time to query local system time and update the timestamp. 

	TON_Time(IN:= TRUE, PT:=T#1200MS ) ; 
	FB_LocalSystTime(
		bEnable := TRUE,
		dwCycle := 1,
		systemTime => CalLocalTimeStruct_Temp);

	IF TON_Time.Q THEN 
		CalLocalTimeStruct:= CalLocalTimeStruct_Temp ; 
	END_IF
	
	FB_ToGMT(
		in	:= CalLocalTimeStruct,
		tzInfo := CstTimeZone_G,
		out	=> CalGMTTimeStruct);
	
	sTimeGMT_G	:= SYSTEMTIME_TO_STRING(CalGMTTimeStruct);
	sTimeLocal_G	:= SYSTEMTIME_TO_STRING(CalLocalTimeStruct);	

////////// 
// The Master PLC takes cpontrol of the power plant , if it is working and has IEC 104 connection working 
// The Slave PLC takles control if PLC master is not responding or if PLC master does not have IEC 104 working . 
////////// 

TON_Stable( IN:= NOT ParamDisablePLCMaster , PT:= ParamStableOP ) ; // Allow time for the master to read slave data after restart
CalStableOp_G :=  TON_Stable.Q ; 


////////////////////// CODE //////////////////////////////////

// INPUTS //
	PRG_IO.M_Inputs() ;  // Refresh DI and AI 
//	ModbusTcp();	// Update modbus TCP server 

//HMI();
	
IF (CstPLCBackup AND (NOT FB_MasterBAckup.bHeartBeat )AND CalStableOp_G) OR (NOT CstPLCBackup AND CalStableOp_G ) OR ParamForceRun  THEN 
// Allow commands, setpoint and orders . 
	OUT_CalRunningPLC_IO := TRUE ; 
// Update redundancy data 
//	Redundancy.M_GetRedundancyData() ; 

ELSIF FB_MasterBAckup.bHeartBeat THEN 
	// Inhib Setpoints and order
	// GET REDUNDANCY DATA FROM DATA 
//	Redundancy.M_ReadRedundancyData() ; 
	OUT_CalRunningPLC_IO := FALSE ; 
ELSE
	
	OUT_CalRunningPLC_IO := FALSE ; 
END_IF 

	A1_PP();

	//PRG_AnnexesFunctions() ; 		// PENSER A DESACTIVER LES ENVOIS DE EMAILS SI REDONDANCE
	//OPC UA 
		OpcUa();
		
// ANALYSIS
	//Analysis();
	
// IO 
	PRG_IO() ; 

// OUTPUTS // 
	PRG_IO.M_Outputs() ;  // Assign DO and AO 

// Database //
	SavePersistent() ;  

//  Au besoin pour inhiber les commandes digitales et les commandes com . 
	R_TRIG_Run(CLK:= OUT_CalRunningPLC_IO) ; 
	F_TRIG_Run(CLK:= OUT_CalRunningPLC_IO) ; 

IF F_TRIG_Run.Q THEN 
	OpcUA.AllDataWPulse.CmdInhibAllWrite 	:= TRUE ; 	// 
	OpcUA.AllDataWPulse.CmdInhibAllRead 	:= TRUE ; 	


ELSIF R_TRIG_Run.Q   THEN 
	IF NOT ParamTest THEN 
		OpcUA.AllDataWPulse.CmdAllowAllWrite	:= TRUE ; 	// Peux ton limiter la réautorization de toutes les ecritures meme si cela avait été forcé à la main auparavant ? 
	END_IF
	OpcUA.AllDataWPulse.CmdAllowAllRead 	:= TRUE ; 	
END_IF

METHOD M_Init : BOOL
VAR_INPUT
END_VAR

VAR 
	Year : STRING ; 
	Month: STRING ; 
	Day : STRING ; 
	Hour: STRING ; 
	Str_Temp: STRING;
END_VAR
//CstCycleTime_G 		:= 50 ;							// Cycle Time
CstTimeZone_G 		:= WEST_EUROPE_TZI ; 		// Local Time Zone 
//Redundancy.M_Init();	



// Get the Windows time ( not accurate ) at startup before updating the system time. 
	// DateTime 
	
	
	FB_GetSystemTime(
		timeLoDW	=> fileTime.dwLowDateTime, 
		timeHiDW	=> fileTime.dwHighDateTime);
		
	FB_ToLocal(
		in			:=fileTime,
		tzInfo 		:= CstTimeZone_G,
		out		 	=> FileTimeLocal);
		
CalLocalTimeStruct := FILETIME_TO_SYSTEMTIME(FileTimelocal) ; 


Year := CONCAT(STR1:= WORD_TO_STRING(CalLocalTimeStruct.wYear), STR2:= '_') ; 
Month := CONCAT(STR1:= WORD_TO_STRING(CalLocalTimeStruct.wMonth), STR2:= '_') ;
Day := CONCAT(STR1:=WORD_TO_STRING(CalLocalTimeStruct.wDay), STR2:= ' ') ;
Hour := CONCAT(STR1:=WORD_TO_STRING(CalLocalTimeStruct.wHour), STR2:= 'h') ;

Str_Temp := Year ; 
Str_Temp := CONCAT(STR1:=Str_Temp , STR2:= Month )  ; 
Str_Temp := CONCAT(STR1:=Str_Temp , STR2:= Day )  ; 	
Str_Temp := CONCAT(STR1:=Str_Temp , STR2:= Hour )  ; 

A1_PP.MesData.MesStartTime 		:= Str_Temp  ; 	// Jour du dernier update de code .
END_METHOD

END_PROGRAM

// ---- 04_Application/IO/PRG_IO.TcPOU
PROGRAM PRG_IO
///////////
// This Program is used as an interface between code variable and the I/O cards
//////////
VAR_INPUT
	
//PP States //
	MesCouplerStatePTR			: ARRAY[1..CstNbPTR_G] OF ST_AI ;

// EXECUTE VARIABLES //
	IN_CmdInhibOutput_OPC		: BOOL := TRUE ; 
	
END_VAR
VAR 	
	MesData				: IO ; 
//M_INIT VARIABLES //
	bInit						: BOOL	:=TRUE ;			// Initialization variables
	iTest                       : INT;
	
	// WAGO Only 
		(*
	xEnable				: 	BOOL := TRUE;
	axDO				: 	ARRAY [1..FR_AppScanKbus.ParameterList_FR_AppScanKbus.MAX_NUMBER_DO] OF BOOL;
	aiAO				: 	ARRAY [1..FR_AppScanKbus.ParameterList_FR_AppScanKbus.MAX_NUMBER_AO] OF INT;
	axDI				: 	ARRAY [1..FR_AppScanKbus.ParameterList_FR_AppScanKbus.MAX_NUMBER_DI] OF BOOL;
	aiAI				: 	ARRAY [1..FR_AppScanKbus.ParameterList_FR_AppScanKbus.MAX_NUMBER_AI] OF INT;
	uiNumberOfModules	: 	UINT;
	atypModule			: 	ARRAY [1..FR_AppScanKbus.ParameterList_FR_AppScanKbus.MAX_NUMBER_OF_MODULES] OF FR_AppScanKbus.typModule;
	xBusy				:	BOOL;
	xError				: 	BOOL;
	sStatus				: 	STRING;
	xKbusInit			: 	BOOL;
	uiNumberOfDO		: 	UINT;
	uiNumberOfDI		: 	UINT;
	uiNumberOfAO		: 	UINT;
	uiNumberOfAI		: 	UINT;
	*)

END_VAR

// Initializing the static variables //  
	IF bInit OR CmdInit_G THEN
		M_Init() ; 
		bInit		:= FALSE ; 
		
	END_IF
	M_AlarmManagement() ; 

	(* WAGO Application
	M_Evaluate() ; 
	
	
FR_AppScanKbus.PRG_ScanKbus(
	xEnable				:= xEnable, 
	axDO				:= axDO, 
	aiAO				:= aiAO, 
	axDI				=> axDI, 
	aiAI				=> aiAI, 
	uiNumberOfModules	=> uiNumberOfModules, 
	atypModule			=> atypModule, 
	xBusy				=> xBusy, 
	xError				=> xError, 
	sStatus				=> sStatus, 
	xKbusInit			=> xKbusInit, 
	uiNumberOfDO		=> uiNumberOfDO, 
	uiNumberOfDI		=> uiNumberOfDI, 
	uiNumberOfAO		=> uiNumberOfAO, 
	uiNumberOfAI		=> uiNumberOfAI, 
	tRefresh			:= T#10MS);
	*)

METHOD M_AlarmManagement
//////////////////
// Generates object alarms and manages resets. 
//////////////////

VAR 
	// Method local variables (reinitialized at each cycle) 
	FB_AlarmCodeManager			: FB_AlarmCodeManager ; 

END_VAR
END_METHOD

METHOD M_Evaluate : BOOL
(*
MesIO_SUBMV_EL1809_1[1].value := axDI[1] ;
MesIO_SUBMV_EL1809_1[2].value := axDI[2] ;
MesIO_SUBMV_EL1809_1[3].value := axDI[3] ;
MesIO_SUBMV_EL1809_1[4].value := axDI[4] ;
MesIO_SUBMV_EL1809_1[5].value := axDI[5] ;
MesIO_SUBMV_EL1809_1[6].value := axDI[6] ;
MesIO_SUBMV_EL1809_1[7].value := axDI[7] ;
MesIO_SUBMV_EL1809_1[8].value := axDI[8] ;
MesIO_SUBMV_EL1809_1[9].value := axDI[9] ;
MesIO_SUBMV_EL1809_1[10].value := axDI[10] ;
MesIO_SUBMV_EL1809_1[11].value := axDI[11] ;
MesIO_SUBMV_EL1809_1[12].value := axDI[12] ;
MesIO_SUBMV_EL1809_1[13].value := axDI[13] ;
MesIO_SUBMV_EL1809_1[14].value := axDI[14] ;
MesIO_SUBMV_EL1809_1[15].value := axDI[15] ;
MesIO_SUBMV_EL1809_1[16].value := axDI[16] ;
MesIO_SUBMV_EL1809_2[1].value := axDI[17] ;
MesIO_SUBMV_EL1809_2[2].value := axDI[18] ;
MesIO_SUBMV_EL1809_2[3].value := axDI[19] ;
MesIO_SUBMV_EL1809_2[4].value := axDI[20] ;
MesIO_SUBMV_EL1809_2[5].value := axDI[21] ;
MesIO_SUBMV_EL1809_2[6].value := axDI[22] ;
MesIO_SUBMV_EL1809_2[7].value := axDI[23] ;
MesIO_SUBMV_EL1809_2[8].value := axDI[24] ;
MesIO_SUBMV_EL1809_2[9].value := axDI[25] ;
MesIO_SUBMV_EL1809_2[10].value := axDI[26] ;
MesIO_SUBMV_EL1809_2[11].value := axDI[27] ;
MesIO_SUBMV_EL1809_2[12].value := axDI[28] ;
MesIO_SUBMV_EL1809_2[13].value := axDI[29] ;
MesIO_SUBMV_EL1809_2[14].value := axDI[30] ;
MesIO_SUBMV_EL1809_2[15].value := axDI[31] ;
MesIO_SUBMV_EL1809_2[16].value := axDI[32] ;
MesIO_SUBMV_EL1809_3[1].value := axDI[33] ;
MesIO_SUBMV_EL1809_3[2].value := axDI[34] ;
MesIO_SUBMV_EL1809_3[3].value := axDI[35] ;
MesIO_SUBMV_EL1809_3[4].value := axDI[36] ;
MesIO_SUBMV_EL1809_3[5].value := axDI[37] ;
MesIO_SUBMV_EL1809_3[6].value := axDI[38] ;
MesIO_SUBMV_EL1809_3[7].value := axDI[39] ;
MesIO_SUBMV_EL1809_3[8].value := axDI[40] ;
MesIO_SUBMV_EL1809_3[9].value := axDI[41] ;
MesIO_SUBMV_EL1809_3[10].value := axDI[42] ;
MesIO_SUBMV_EL1809_3[11].value := axDI[43] ;
MesIO_SUBMV_EL1809_3[12].value := axDI[44] ;
MesIO_SUBMV_EL1809_3[13].value := axDI[45] ;
MesIO_SUBMV_EL1809_3[14].value := axDI[46] ;
MesIO_SUBMV_EL1809_3[15].value := axDI[47] ;
MesIO_SUBMV_EL1809_3[16].value := axDI[48] ;
axDO[1] := MesIO_SUBMV_EL2809_4[1].value ; 
axDO[2] := MesIO_SUBMV_EL2809_4[2].value ; 
axDO[3] := MesIO_SUBMV_EL2809_4[3].value ; 
axDO[4] := MesIO_SUBMV_EL2809_4[4].value ; 
axDO[5] := MesIO_SUBMV_EL2809_4[5].value ; 
axDO[6] := MesIO_SUBMV_EL2809_4[6].value ; 
axDO[7] := MesIO_SUBMV_EL2809_4[7].value ; 
axDO[8] := MesIO_SUBMV_EL2809_4[8].value ; 
axDO[9] := MesIO_SUBMV_EL2809_4[9].value ; 
axDO[10] := MesIO_SUBMV_EL2809_4[10].value ; 
axDO[11] := MesIO_SUBMV_EL2809_4[11].value ; 
axDO[12] := MesIO_SUBMV_EL2809_4[12].value ; 
axDO[13] := MesIO_SUBMV_EL2809_4[13].value ; 
axDO[14] := MesIO_SUBMV_EL2809_4[14].value ; 
axDO[15] := MesIO_SUBMV_EL2809_4[15].value ; 
axDO[16] := MesIO_SUBMV_EL2809_4[16].value ; 
MesIO_SUBMV_EL3024_5[1].value := axAI[1] ;
MesIO_SUBMV_EL3024_5[2].value := axAI[2] ;
MesIO_SUBMV_EL3024_5[3].value := axAI[3] ;
MesIO_SUBMV_EL3024_5[4].value := axAI[4] ;
MesIO_PTR_1_EL3024_8[1].value := axAI[5] ;
MesIO_PTR_1_EL3024_8[2].value := axAI[6] ;
MesIO_PTR_1_EL3024_8[3].value := axAI[7] ;
MesIO_PTR_1_EL3024_8[4].value := axAI[8] ;
MesIO_PTR_1_EL1809_9[1].value := axDI[49] ;
MesIO_PTR_1_EL1809_9[2].value := axDI[50] ;
MesIO_PTR_1_EL1809_9[3].value := axDI[51] ;
MesIO_PTR_1_EL1809_9[4].value := axDI[52] ;
MesIO_PTR_1_EL1809_9[5].value := axDI[53] ;
MesIO_PTR_1_EL1809_9[6].value := axDI[54] ;
MesIO_PTR_1_EL1809_9[7].value := axDI[55] ;
MesIO_PTR_1_EL1809_9[8].value := axDI[56] ;
MesIO_PTR_1_EL1809_9[9].value := axDI[57] ;
MesIO_PTR_1_EL1809_9[10].value := axDI[58] ;
MesIO_PTR_1_EL1809_9[11].value := axDI[59] ;
MesIO_PTR_1_EL1809_9[12].value := axDI[60] ;
MesIO_PTR_1_EL1809_9[13].value := axDI[61] ;
MesIO_PTR_1_EL1809_9[14].value := axDI[62] ;
MesIO_PTR_1_EL1809_9[15].value := axDI[63] ;
MesIO_PTR_1_EL1809_9[16].value := axDI[64] ;
axDO[17] := MesIO_PTR_1_EL2809_10[1].value ; 
axDO[18] := MesIO_PTR_1_EL2809_10[2].value ; 
axDO[19] := MesIO_PTR_1_EL2809_10[3].value ; 
axDO[20] := MesIO_PTR_1_EL2809_10[4].value ; 
axDO[21] := MesIO_PTR_1_EL2809_10[5].value ; 
axDO[22] := MesIO_PTR_1_EL2809_10[6].value ; 
axDO[23] := MesIO_PTR_1_EL2809_10[7].value ; 
axDO[24] := MesIO_PTR_1_EL2809_10[8].value ; 
axDO[25] := MesIO_PTR_1_EL2809_10[9].value ; 
axDO[26] := MesIO_PTR_1_EL2809_10[10].value ; 
axDO[27] := MesIO_PTR_1_EL2809_10[11].value ; 
axDO[28] := MesIO_PTR_1_EL2809_10[12].value ; 
axDO[29] := MesIO_PTR_1_EL2809_10[13].value ; 
axDO[30] := MesIO_PTR_1_EL2809_10[14].value ; 
axDO[31] := MesIO_PTR_1_EL2809_10[15].value ; 
axDO[32] := MesIO_PTR_1_EL2809_10[16].value ; 
MesIO_PTR_2_EL3024_8[1].value := axAI[9] ;
MesIO_PTR_2_EL3024_8[2].value := axAI[10] ;
MesIO_PTR_2_EL3024_8[3].value := axAI[11] ;
MesIO_PTR_2_EL3024_8[4].value := axAI[12] ;
MesIO_PTR_2_EL1809_9[1].value := axDI[65] ;
MesIO_PTR_2_EL1809_9[2].value := axDI[66] ;
MesIO_PTR_2_EL1809_9[3].value := axDI[67] ;
MesIO_PTR_2_EL1809_9[4].value := axDI[68] ;
MesIO_PTR_2_EL1809_9[5].value := axDI[69] ;
MesIO_PTR_2_EL1809_9[6].value := axDI[70] ;
MesIO_PTR_2_EL1809_9[7].value := axDI[71] ;
MesIO_PTR_2_EL1809_9[8].value := axDI[72] ;
MesIO_PTR_2_EL1809_9[9].value := axDI[73] ;
MesIO_PTR_2_EL1809_9[10].value := axDI[74] ;
MesIO_PTR_2_EL1809_9[11].value := axDI[75] ;
MesIO_PTR_2_EL1809_9[12].value := axDI[76] ;
MesIO_PTR_2_EL1809_9[13].value := axDI[77] ;
MesIO_PTR_2_EL1809_9[14].value := axDI[78] ;
MesIO_PTR_2_EL1809_9[15].value := axDI[79] ;
MesIO_PTR_2_EL1809_9[16].value := axDI[80] ;
axDO[33] := MesIO_PTR_2_EL2809_10[1].value ; 
axDO[34] := MesIO_PTR_2_EL2809_10[2].value ; 
axDO[35] := MesIO_PTR_2_EL2809_10[3].value ; 
axDO[36] := MesIO_PTR_2_EL2809_10[4].value ; 
axDO[37] := MesIO_PTR_2_EL2809_10[5].value ; 
axDO[38] := MesIO_PTR_2_EL2809_10[6].value ; 
axDO[39] := MesIO_PTR_2_EL2809_10[7].value ; 
axDO[40] := MesIO_PTR_2_EL2809_10[8].value ; 
axDO[41] := MesIO_PTR_2_EL2809_10[9].value ; 
axDO[42] := MesIO_PTR_2_EL2809_10[10].value ; 
axDO[43] := MesIO_PTR_2_EL2809_10[11].value ; 
axDO[44] := MesIO_PTR_2_EL2809_10[12].value ; 
axDO[45] := MesIO_PTR_2_EL2809_10[13].value ; 
axDO[46] := MesIO_PTR_2_EL2809_10[14].value ; 
axDO[47] := MesIO_PTR_2_EL2809_10[15].value ; 
axDO[48] := MesIO_PTR_2_EL2809_10[16].value ; 
MesIO_PTR_3_EL3024_8[1].value := axAI[13] ;
MesIO_PTR_3_EL3024_8[2].value := axAI[14] ;
MesIO_PTR_3_EL3024_8[3].value := axAI[15] ;
MesIO_PTR_3_EL3024_8[4].value := axAI[16] ;
MesIO_PTR_3_EL1809_9[1].value := axDI[81] ;
MesIO_PTR_3_EL1809_9[2].value := axDI[82] ;
MesIO_PTR_3_EL1809_9[3].value := axDI[83] ;
MesIO_PTR_3_EL1809_9[4].value := axDI[84] ;
MesIO_PTR_3_EL1809_9[5].value := axDI[85] ;
MesIO_PTR_3_EL1809_9[6].value := axDI[86] ;
MesIO_PTR_3_EL1809_9[7].value := axDI[87] ;
MesIO_PTR_3_EL1809_9[8].value := axDI[88] ;
MesIO_PTR_3_EL1809_9[9].value := axDI[89] ;
MesIO_PTR_3_EL1809_9[10].value := axDI[90] ;
MesIO_PTR_3_EL1809_9[11].value := axDI[91] ;
MesIO_PTR_3_EL1809_9[12].value := axDI[92] ;
MesIO_PTR_3_EL1809_9[13].value := axDI[93] ;
MesIO_PTR_3_EL1809_9[14].value := axDI[94] ;
MesIO_PTR_3_EL1809_9[15].value := axDI[95] ;
MesIO_PTR_3_EL1809_9[16].value := axDI[96] ;
axDO[49] := MesIO_PTR_3_EL2809_10[1].value ; 
axDO[50] := MesIO_PTR_3_EL2809_10[2].value ; 
axDO[51] := MesIO_PTR_3_EL2809_10[3].value ; 
axDO[52] := MesIO_PTR_3_EL2809_10[4].value ; 
axDO[53] := MesIO_PTR_3_EL2809_10[5].value ; 
axDO[54] := MesIO_PTR_3_EL2809_10[6].value ; 
axDO[55] := MesIO_PTR_3_EL2809_10[7].value ; 
axDO[56] := MesIO_PTR_3_EL2809_10[8].value ; 
axDO[57] := MesIO_PTR_3_EL2809_10[9].value ; 
axDO[58] := MesIO_PTR_3_EL2809_10[10].value ; 
axDO[59] := MesIO_PTR_3_EL2809_10[11].value ; 
axDO[60] := MesIO_PTR_3_EL2809_10[12].value ; 
axDO[61] := MesIO_PTR_3_EL2809_10[13].value ; 
axDO[62] := MesIO_PTR_3_EL2809_10[14].value ; 
axDO[63] := MesIO_PTR_3_EL2809_10[15].value ; 
axDO[64] := MesIO_PTR_3_EL2809_10[16].value ; 
*)
END_METHOD

METHOD M_Init : BOOL
VAR
	KK : BYTE;
END_VAR
END_METHOD

METHOD M_Inputs
///////////
// Intput interface between POUs and I/O Cards
//////////////

VAR 
KK							: BYTE ; 					// For LOOP 
MesCouplerStateSUB_MV			: ST_AI ; 
END_VAR
END_METHOD

METHOD M_Outputs : BOOL
///////////
// Intput interface between POUs and I/O Cards
//////////////
VAR
	KK	: BYTE;

	A1_MainMVCB: INT;
END_VAR
END_METHOD

END_PROGRAM

